KUKA KRL program: MyProgram_165().src

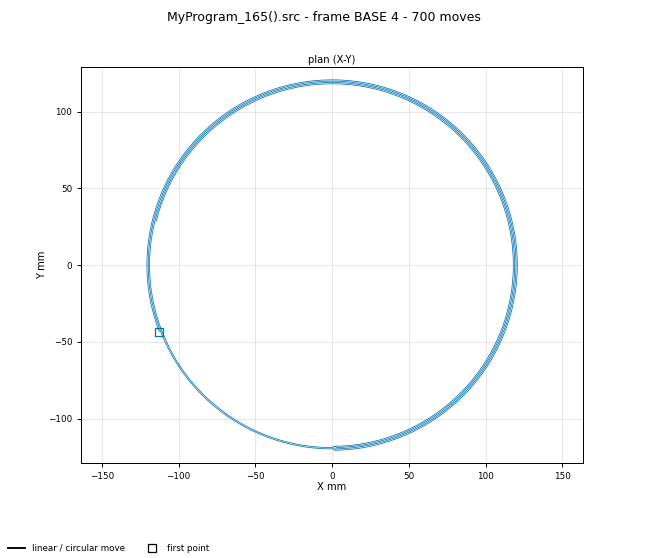
[picture p0: tool path of MyProgram_165().src in frame BASE 4, 700 of 700 moves have a stored position in this frame; points joined in program order, loops and branches not executed]
&ACCESS RVP
&REL 1
&PARAM TEMPLATE = C:\KRC\Roboter\Template\vorgabe
&PARAM EDITMASK = *
DEF MyProgram_165()
; ---- Setting reference (Base) ----
$BASE = BASE_DATA[4]

; --------------------------
; ---- Setting tool (TCP) ----
$TOOL = TOOL_DATA[3]
; --------------------------

$VEL.CP = VEL_APROX_PRINT
Startdeposition()
$VEL.CP = VEL_PRINT
LIN {X -112.6029,Y -43.4357,Z 125,A -162.8947,B 24.9558,C -1.5362,E1 24.8502,E2 249.1159} C_DIS
LIN {X -113.6349,Y -40.6592,Z 125,A -164.31,B 24.9556,C -1.54,E1 24.8489,E2 250.5301} C_DIS
LIN {X -114.5985,Y -37.8582,Z 125,A -165.7254,B 24.9553,C -1.5438,E1 24.8476,E2 251.9444} C_DIS
LIN {X -115.4923,Y -35.0371,Z 125,A -167.1395,B 24.9551,C -1.5477,E1 24.8464,E2 253.3573} C_DIS
LIN {X -116.1833,Y -32.6652,Z 125,A -168.3736,B 24.9551,C -1.5488,E1 24.8455,E2 254.5961} C_DIS
LIN {X -117.0731,Y -29.3253,Z 125,A -169.9721,B 24.9547,C -1.5556,E1 24.8444,E2 256.1875} C_DIS
LIN {X -117.7575,Y -26.4433,Z 125,A -171.3879,B 24.9544,C -1.5596,E1 24.8435,E2 257.6022} C_DIS
LIN {X -118.371,Y -23.5454,Z 125,A -172.8035,B 24.9542,C -1.5637,E1 24.8427,E2 259.0165} C_DIS
LIN {X -118.9131,Y -20.6334,Z 125,A -174.2195,B 24.954,C -1.5677,E1 24.842,E2 260.4313} C_DIS
LIN {X -119.592,Y -16.2425,Z 125,A -176.3434,B 24.9536,C -1.5738,E1 24.8411,E2 262.5532} C_DIS
LIN {X -119.9546,Y -13.3027,Z 125,A -177.7592,B 24.9533,C -1.578,E1 24.8407,E2 263.9677} C_DIS
LIN {X -120.2449,Y -10.3549,Z 125,A -179.1753,B 24.9531,C -1.5821,E1 24.8403,E2 265.3825} C_DIS
LIN {X -120.4629,Y -7.4008,Z 125,A 179.4086,B 24.9529,C -1.5862,E1 24.84,E2 266.7971} C_DIS
LIN {X -120.6082,Y -4.4423,Z 125,A 177.9925,B 24.9526,C -1.5904,E1 24.8399,E2 268.2119} C_DIS
LIN {X -120.6878,Y -0.4383,Z 125,A 176.0198,B 24.9524,C -1.5936,E1 24.8398,E2 270.1888} C_DIS
LIN {X -120.6536,Y 2.9619,Z 125,A 174.4521,B 24.952,C -1.6008,E1 24.8398,E2 271.7488} C_DIS
LIN {X -120.5446,Y 5.922,Z 125,A 173.0359,B 24.9517,C -1.605,E1 24.84,E2 273.1636} C_DIS
LIN {X -120.363,Y 8.8785,Z 125,A 171.6198,B 24.9515,C -1.6091,E1 24.8403,E2 274.5783} C_DIS
LIN {X -120.1088,Y 11.8297,Z 125,A 170.2037,B 24.9512,C -1.6133,E1 24.8407,E2 275.9929} C_DIS
LIN {X -119.7823,Y 14.7737,Z 125,A 168.7876,B 24.951,C -1.6175,E1 24.8411,E2 277.4075} C_DIS
LIN {X -119.2402,Y 18.6372,Z 125,A 166.8598,B 24.9508,C -1.6204,E1 24.8419,E2 279.34} C_DIS
LIN {X -118.651,Y 22.0911,Z 125,A 165.2473,B 24.9503,C -1.6279,E1 24.8427,E2 280.9441} C_DIS
LIN {X -118.0731,Y 24.9963,Z 125,A 163.8312,B 24.9501,C -1.632,E1 24.8435,E2 282.3587} C_DIS
LIN {X -117.4241,Y 27.8864,Z 125,A 162.4152,B 24.9498,C -1.6361,E1 24.8444,E2 283.7732} C_DIS
LIN {X -116.7044,Y 30.7597,Z 125,A 160.9991,B 24.9496,C -1.6402,E1 24.8453,E2 285.1878} C_DIS
LIN {X -115.9143,Y 33.6145,Z 125,A 159.5832,B 24.9493,C -1.6443,E1 24.8464,E2 286.6021} C_DIS
LIN {X -115.1524,Y 36.1334,Z 125,A 158.2993,B 24.9492,C -1.6468,E1 24.8475,E2 287.8873} C_DIS
LIN {X -114.1253,Y 39.2617,Z 125,A 156.7515,B 24.9488,C -1.6524,E1 24.8488,E2 289.4308} C_DIS
LIN {X -113.1274,Y 42.0506,Z 125,A 155.3357,B 24.9486,C -1.6564,E1 24.8502,E2 290.8451} C_DIS
LIN {X -112.0614,Y 44.8143,Z 125,A 153.9202,B 24.9483,C -1.6604,E1 24.8516,E2 292.259} C_DIS
LIN {X -110.9278,Y 47.5509,Z 125,A 152.5045,B 24.9481,C -1.6643,E1 24.8532,E2 293.6731} C_DIS
LIN {X -109.7275,Y 50.2589,Z 125,A 151.089,B 24.9478,C -1.6682,E1 24.8548,E2 295.0871} C_DIS
LIN {X -108.461,Y 52.9366,Z 125,A 149.6737,B 24.9476,C -1.6721,E1 24.8565,E2 296.5009} C_DIS
LIN {X -107.1292,Y 55.5824,Z 125,A 148.2584,B 24.9474,C -1.6759,E1 24.8583,E2 297.9146} C_DIS
LIN {X -105.7329,Y 58.1948,Z 125,A 146.8429,B 24.9471,C -1.6797,E1 24.8602,E2 299.3286} C_DIS
LIN {X -104.2729,Y 60.772,Z 125,A 145.4281,B 24.9469,C -1.6835,E1 24.8621,E2 300.7418} C_DIS
LIN {X -102.75,Y 63.3127,Z 125,A 144.013,B 24.9467,C -1.6871,E1 24.8642,E2 302.1554} C_DIS
LIN {X -101.1653,Y 65.8153,Z 125,A 142.598,B 24.9464,C -1.6908,E1 24.8663,E2 303.5688} C_DIS
LIN {X -99.5197,Y 68.2782,Z 125,A 141.1833,B 24.9462,C -1.6944,E1 24.8685,E2 304.9821} C_DIS
LIN {X -97.8985,Y 70.5815,Z 125,A 139.8326,B 24.946,C -1.6975,E1 24.8707,E2 306.3319} C_DIS
LIN {X -96.0495,Y 73.0791,Z 125,A 138.3539,B 24.9458,C -1.7014,E1 24.8732,E2 307.8084} C_DIS
LIN {X -93.2946,Y 76.5649,Z 125,A 136.233,B 24.9454,C -1.7065,E1 24.8769,E2 309.9271} C_DIS
LIN {X -91.3875,Y 78.8314,Z 125,A 134.8186,B 24.9452,C -1.7099,E1 24.8794,E2 311.34} C_DIS
LIN {X -89.4254,Y 81.0504,Z 125,A 133.4045,B 24.945,C -1.7131,E1 24.8821,E2 312.7527} C_DIS
LIN {X -87.4094,Y 83.2206,Z 125,A 131.9907,B 24.9448,C -1.7163,E1 24.8848,E2 314.1649} C_DIS
LIN {X -85.3407,Y 85.3407,Z 125,A 130.577,B 24.9446,C -1.7195,E1 24.8875,E2 315.5772} C_DIS
LIN {X -83.2206,Y 87.4094,Z 125,A 129.1635,B 24.9444,C -1.7225,E1 24.8904,E2 316.9892} C_DIS
LIN {X -81.0504,Y 89.4254,Z 125,A 127.7501,B 24.9442,C -1.7255,E1 24.8933,E2 318.4012} C_DIS
LIN {X -78.8314,Y 91.3875,Z 125,A 126.3371,B 24.944,C -1.7285,E1 24.8963,E2 319.8128} C_DIS
LIN {X -76.5649,Y 93.2946,Z 125,A 124.9241,B 24.9438,C -1.7313,E1 24.8993,E2 321.2244} C_DIS
LIN {X -74.2523,Y 95.1455,Z 125,A 123.511,B 24.9436,C -1.7341,E1 24.9024,E2 322.6362} C_DIS
LIN {X -71.8949,Y 96.9391,Z 125,A 122.0984,B 24.9435,C -1.7368,E1 24.9055,E2 324.0474} C_DIS
LIN {X -69.4943,Y 98.6743,Z 125,A 120.6859,B 24.9433,C -1.7394,E1 24.9087,E2 325.4586} C_DIS
LIN {X -67.0518,Y 100.3501,Z 125,A 119.2737,B 24.9431,C -1.742,E1 24.912,E2 326.8695} C_DIS
LIN {X -63.7759,Y 102.4607,Z 125,A 117.3526,B 24.9431,C -1.7425,E1 24.9165,E2 328.7955} C_DIS
LIN {X -60.772,Y 104.2729,Z 125,A 115.744,B 24.9427,C -1.7479,E1 24.9204,E2 330.396} C_DIS
LIN {X -57.2872,Y 106.2252,Z 125,A 113.8456,B 24.9425,C -1.7512,E1 24.925,E2 332.292} C_DIS
LIN {X -54.2636,Y 107.8032,Z 125,A 112.2154,B 24.9424,C -1.7534,E1 24.9291,E2 333.9215} C_DIS
LIN {X -51.6016,Y 109.1025,Z 125,A 110.804,B 24.9422,C -1.7554,E1 24.9326,E2 335.3317} C_DIS
LIN {X -48.1374,Y 110.6722,Z 125,A 108.9928,B 24.9421,C -1.7579,E1 24.9372,E2 337.1413} C_DIS
LIN {X -45.4069,Y 111.8202,Z 125,A 107.5823,B 24.942,C -1.7597,E1 24.9409,E2 338.5507} C_DIS
LIN {X -42.3982,Y 112.9958,Z 125,A 106.0121,B 24.942,C -1.7602,E1 24.945,E2 340.1232} C_DIS
LIN {X -39.2617,Y 114.1253,Z 125,A 104.4574,B 24.9417,C -1.7634,E1 24.949,E2 341.6733} C_DIS
LIN {X -36.4491,Y 115.0545,Z 125,A 103.0473,B 24.9417,C -1.7649,E1 24.9528,E2 343.0823} C_DIS
LIN {X -33.6145,Y 115.9143,Z 125,A 101.6376,B 24.9415,C -1.7663,E1 24.9566,E2 344.491} C_DIS
LIN {X -30.7597,Y 116.7044,Z 125,A 100.2283,B 24.9415,C -1.7676,E1 24.9604,E2 345.8993} C_DIS
LIN {X -27.8864,Y 117.4241,Z 125,A 98.8194,B 24.9414,C -1.7689,E1 24.9642,E2 347.3072} C_DIS
LIN {X -24.9963,Y 118.0731,Z 125,A 97.4103,B 24.9413,C -1.77,E1 24.968,E2 348.7155} C_DIS
LIN {X -22.0911,Y 118.651,Z 125,A 96.0017,B 24.9413,C -1.771,E1 24.9719,E2 350.1232} C_DIS
LIN {X -18.3412,Y 119.2859,Z 125,A 94.2227,B 24.941,C -1.7736,E1 24.9768,E2 351.8978} C_DIS
LIN {X -15.4082,Y 119.7001,Z 125,A 92.7653,B 24.9411,C -1.7722,E1 24.9808,E2 353.3596} C_DIS
LIN {X -11.8297,Y 120.1088,Z 125,A 91.073,B 24.9411,C -1.7738,E1 24.9855,E2 355.0489} C_DIS
LIN {X -8.8785,Y 120.363,Z 125,A 89.6655,B 24.941,C -1.7744,E1 24.9894,E2 356.4557} C_DIS
LIN {X -5.922,Y 120.5446,Z 125,A 88.2578,B 24.941,C -1.7749,E1 24.9933,E2 357.8628} C_DIS
LIN {X -1.4811,Y 120.6809,Z 125,A 86.1474,B 24.941,C -1.7754,E1 24.9992,E2 359.9721} C_DIS
LIN {X 1.4811,Y 120.6809,Z 125,A 84.7407,B 24.941,C -1.7757,E1 25.0032,E2 361.3781} C_DIS
LIN {X 4.4423,Y 120.6082,Z 125,A 83.3343,B 24.9409,C -1.7757,E1 25.0071,E2 362.784} C_DIS
LIN {X 7.4008,Y 120.4629,Z 125,A 81.9278,B 24.9409,C -1.7757,E1 25.011,E2 364.1899} C_DIS
LIN {X 10.3549,Y 120.2449,Z 125,A 80.5218,B 24.9409,C -1.7757,E1 25.0149,E2 365.5953} C_DIS
LIN {X 13.3027,Y 119.9546,Z 125,A 79.116,B 24.9409,C -1.7755,E1 25.0188,E2 367.0006} C_DIS
LIN {X 16.2425,Y 119.592,Z 125,A 77.7102,B 24.9409,C -1.7752,E1 25.0227,E2 368.4061} C_DIS
LIN {X 19.1726,Y 119.1574,Z 125,A 76.3051,B 24.9409,C -1.7748,E1 25.0266,E2 369.8107} C_DIS
LIN {X 22.0911,Y 118.651,Z 125,A 74.8999,B 24.9409,C -1.7744,E1 25.0304,E2 371.2155} C_DIS
LIN {X 24.9963,Y 118.0731,Z 125,A 73.4952,B 24.941,C -1.7738,E1 25.0343,E2 372.6198} C_DIS
LIN {X 27.8864,Y 117.4241,Z 125,A 72.0905,B 24.941,C -1.7731,E1 25.0381,E2 374.0243} C_DIS
LIN {X 30.7597,Y 116.7044,Z 125,A 70.6861,B 24.9411,C -1.7723,E1 25.0419,E2 375.4284} C_DIS
LIN {X 33.6145,Y 115.9143,Z 125,A 69.2821,B 24.9411,C -1.7714,E1 25.0457,E2 376.8321} C_DIS
LIN {X 36.4491,Y 115.0545,Z 125,A 67.878,B 24.9413,C -1.7704,E1 25.0494,E2 378.236} C_DIS
LIN {X 38.7619,Y 114.2938,Z 125,A 66.6649,B 24.9415,C -1.7668,E1 25.0527,E2 379.4554} C_DIS
LIN {X 42.0506,Y 113.1274,Z 125,A 65.0709,B 24.9415,C -1.7682,E1 25.0568,E2 381.0428} C_DIS
LIN {X 44.8143,Y 112.0614,Z 125,A 63.6677,B 24.9415,C -1.7669,E1 25.0605,E2 382.446} C_DIS
LIN {X 47.5509,Y 110.9278,Z 125,A 62.2648,B 24.9415,C -1.7655,E1 25.0641,E2 383.8488} C_DIS
LIN {X 50.2589,Y 109.7275,Z 125,A 60.8619,B 24.9417,C -1.764,E1 25.0676,E2 385.2517} C_DIS
LIN {X 52.9366,Y 108.461,Z 125,A 59.4596,B 24.9417,C -1.7625,E1 25.0712,E2 386.654} C_DIS
LIN {X 56.562,Y 106.6133,Z 125,A 57.5008,B 24.942,C -1.7587,E1 25.076,E2 388.6164} C_DIS
LIN {X 59.4879,Y 105.0108,Z 125,A 55.954,B 24.942,C -1.7581,E1 25.0798,E2 390.1599} C_DIS
LIN {X 62.0471,Y 103.5193,Z 125,A 54.5523,B 24.9422,C -1.7563,E1 25.0832,E2 391.5618} C_DIS
LIN {X 64.3587,Y 102.0967,Z 125,A 53.2527,B 24.9424,C -1.7538,E1 25.0863,E2 392.8631} C_DIS
LIN {X 67.0518,Y 100.3501,Z 125,A 51.7493,B 24.9424,C -1.7522,E1 25.0898,E2 394.3652} C_DIS
LIN {X 69.4943,Y 98.6743,Z 125,A 50.3482,B 24.9426,C -1.7501,E1 25.093,E2 395.7666} C_DIS
LIN {X 71.6715,Y 97.1027,Z 125,A 49.0595,B 24.9428,C -1.7472,E1 25.0959,E2 397.0575} C_DIS
LIN {X 74.2523,Y 95.1455,Z 125,A 47.5463,B 24.9428,C -1.7455,E1 25.0992,E2 398.5691} C_DIS
LIN {X 76.5649,Y 93.2946,Z 125,A 46.1458,B 24.9431,C -1.7431,E1 25.1023,E2 399.97} C_DIS
LIN {X 78.5212,Y 91.6518,Z 125,A 44.9007,B 24.9433,C -1.7392,E1 25.1049,E2 401.2194} C_DIS
LIN {X 81.0504,Y 89.4254,Z 125,A 43.3453,B 24.9433,C -1.7381,E1 25.1082,E2 402.7713} C_DIS
LIN {X 83.2206,Y 87.4094,Z 125,A 41.9454,B 24.9436,C -1.7354,E1 25.111,E2 404.1718} C_DIS
LIN {X 85.3407,Y 85.3407,Z 125,A 40.5457,B 24.9437,C -1.7327,E1 25.1138,E2 405.572} C_DIS
LIN {X 87.4094,Y 83.2206,Z 125,A 39.146,B 24.9439,C -1.7299,E1 25.1165,E2 406.9723} C_DIS
LIN {X 89.4086,Y 81.0687,Z 125,A 37.758,B 24.9441,C -1.7271,E1 25.1191,E2 408.3609} C_DIS
LIN {X 91.3875,Y 78.8314,Z 125,A 36.3474,B 24.9443,C -1.7241,E1 25.1217,E2 409.7721} C_DIS
LIN {X 93.2946,Y 76.5649,Z 125,A 34.948,B 24.9445,C -1.7211,E1 25.1242,E2 411.1721} C_DIS
LIN {X 95.1455,Y 74.2523,Z 125,A 33.5493,B 24.9447,C -1.718,E1 25.1267,E2 412.5716} C_DIS
LIN {X 96.9391,Y 71.8949,Z 125,A 32.1503,B 24.9449,C -1.7149,E1 25.129,E2 413.9713} C_DIS
LIN {X 98.6743,Y 69.4943,Z 125,A 30.7518,B 24.9451,C -1.7117,E1 25.1313,E2 415.3705} C_DIS
LIN {X 100.3501,Y 67.0518,Z 125,A 29.3533,B 24.9453,C -1.7084,E1 25.1335,E2 416.7699} C_DIS
LIN {X 101.9654,Y 64.5689,Z 125,A 27.9547,B 24.9455,C -1.7051,E1 25.1356,E2 418.1693} C_DIS
LIN {X 103.3302,Y 62.3582,Z 125,A 26.6977,B 24.9458,C -1.7007,E1 25.1374,E2 419.4303} C_DIS
LIN {X 105.0108,Y 59.4879,Z 125,A 25.1587,B 24.946,C -1.6983,E1 25.1396,E2 420.967} C_DIS
LIN {X 106.4391,Y 56.8929,Z 125,A 23.7606,B 24.9462,C -1.6948,E1 25.1414,E2 422.3661} C_DIS
LIN {X 107.8032,Y 54.2636,Z 125,A 22.3629,B 24.9464,C -1.6912,E1 25.1432,E2 423.7647} C_DIS
LIN {X 109.1025,Y 51.6016,Z 125,A 20.9651,B 24.9466,C -1.6876,E1 25.1449,E2 425.1635} C_DIS
LIN {X 110.336,Y 48.9086,Z 125,A 19.5676,B 24.9469,C -1.684,E1 25.1465,E2 426.562} C_DIS
LIN {X 111.503,Y 46.1861,Z 125,A 18.1699,B 24.9471,C -1.6803,E1 25.148,E2 427.9608} C_DIS
LIN {X 112.5558,Y 43.5555,Z 125,A 16.829,B 24.9473,C -1.6765,E1 25.1494,E2 429.3032} C_DIS
LIN {X 113.588,Y 40.788,Z 125,A 15.4352,B 24.9476,C -1.6727,E1 25.1507,E2 430.6981} C_DIS
LIN {X 114.5985,Y 37.8582,Z 125,A 13.978,B 24.9478,C -1.6689,E1 25.152,E2 432.1559} C_DIS
LIN {X 115.4931,Y 35.0344,Z 125,A 12.5811,B 24.948,C -1.6651,E1 25.1532,E2 433.554} C_DIS
LIN {X 116.3181,Y 32.1896,Z 125,A 11.184,B 24.9483,C -1.6612,E1 25.1543,E2 434.9522} C_DIS
LIN {X 117.0731,Y 29.3253,Z 125,A 9.787,B 24.9485,C -1.6573,E1 25.1552,E2 436.3504} C_DIS
LIN {X 117.7575,Y 26.4433,Z 125,A 8.3902,B 24.9488,C -1.6533,E1 25.1561,E2 437.7485} C_DIS
LIN {X 118.371,Y 23.5454,Z 125,A 6.9934,B 24.949,C -1.6493,E1 25.1569,E2 439.1465} C_DIS
LIN {X 118.9131,Y 20.6334,Z 125,A 5.5965,B 24.9493,C -1.6453,E1 25.1576,E2 440.5447} C_DIS
LIN {X 119.3837,Y 17.7089,Z 125,A 4.2001,B 24.9495,C -1.6413,E1 25.1582,E2 441.9423} C_DIS
LIN {X 119.7823,Y 14.7737,Z 125,A 2.8031,B 24.9498,C -1.6372,E1 25.1587,E2 443.3406} C_DIS
LIN {X 120.1088,Y 11.8297,Z 125,A 1.4066,B 24.95,C -1.6332,E1 25.1591,E2 444.7385} C_DIS
LIN {X 120.363,Y 8.8785,Z 125,A 0.0101,B 24.9503,C -1.6291,E1 25.1594,E2 446.1363} C_DIS
LIN {X 120.5446,Y 5.922,Z 125,A -1.3868,B 24.9505,C -1.625,E1 25.1596,E2 447.5346} C_DIS
LIN {X 120.6809,Y 1.481,Z 125,A -3.6105,B 24.9513,C -1.6125,E1 25.1598,E2 449.7746} C_DIS
LIN {X 120.6536,Y -2.9619,Z 125,A -5.5761,B 24.9513,C -1.6127,E1 25.1598,E2 451.728} C_DIS
LIN {X 120.5446,Y -5.922,Z 125,A -6.9725,B 24.9515,C -1.6085,E1 25.1595,E2 453.1259} C_DIS
LIN {X 120.363,Y -8.8785,Z 125,A -8.369,B 24.9518,C -1.6044,E1 25.1593,E2 454.5238} C_DIS
LIN {X 120.1088,Y -11.8297,Z 125,A -9.7654,B 24.952,C -1.6003,E1 25.1589,E2 455.9217} C_DIS
LIN {X 119.7823,Y -14.7737,Z 125,A -11.1618,B 24.9523,C -1.5962,E1 25.1585,E2 457.3195} C_DIS
LIN {X 119.3837,Y -17.7089,Z 125,A -12.5582,B 24.9525,C -1.592,E1 25.1579,E2 458.7173} C_DIS
LIN {X 118.9131,Y -20.6334,Z 125,A -13.955,B 24.9528,C -1.5879,E1 25.1573,E2 460.1156} C_DIS
LIN {X 118.371,Y -23.5454,Z 125,A -15.3514,B 24.953,C -1.5838,E1 25.1565,E2 461.5136} C_DIS
LIN {X 117.5681,Y -27.263,Z 125,A -17.1815,B 24.9534,C -1.5768,E1 25.1554,E2 463.3496} C_DIS
LIN {X 116.7044,Y -30.7597,Z 125,A -18.843,B 24.9536,C -1.5737,E1 25.1543,E2 465.0089} C_DIS
LIN {X 115.9143,Y -33.6145,Z 125,A -20.2397,B 24.9538,C -1.5696,E1 25.1532,E2 466.4072} C_DIS
LIN {X 115.0545,Y -36.4491,Z 125,A -21.6363,B 24.9541,C -1.5656,E1 25.1521,E2 467.8053} C_DIS
LIN {X 114.1253,Y -39.2617,Z 125,A -23.0331,B 24.9543,C -1.5616,E1 25.1508,E2 469.2036} C_DIS
LIN {X 113.1274,Y -42.0506,Z 125,A -24.43,B 24.9545,C -1.5576,E1 25.1495,E2 470.602} C_DIS
LIN {X 112.0614,Y -44.8143,Z 125,A -25.8269,B 24.9548,C -1.5537,E1 25.1481,E2 472.0005} C_DIS
LIN {X 111.1126,Y -47.1124,Z 125,A -27.0487,B 24.9551,C -1.548,E1 25.1467,E2 473.2289} C_DIS
LIN {X 109.7275,Y -50.2589,Z 125,A -28.621,B 24.9552,C -1.5459,E1 25.1449,E2 474.7976} C_DIS
LIN {X 108.5122,Y -52.8301,Z 125,A -29.9662,B 24.9554,C -1.5421,E1 25.1433,E2 476.1447} C_DIS
LIN {X 107.1309,Y -55.5791,Z 125,A -31.4135,B 24.9557,C -1.5383,E1 25.1415,E2 477.5932} C_DIS
LIN {X 105.7329,Y -58.1948,Z 125,A -32.8128,B 24.9559,C -1.5345,E1 25.1396,E2 478.994} C_DIS
LIN {X 104.4838,Y -60.405,Z 125,A -34.0505,B 24.9562,C -1.5294,E1 25.1379,E2 480.2374} C_DIS
LIN {X 102.75,Y -63.3127,Z 125,A -35.6077,B 24.9563,C -1.5271,E1 25.1356,E2 481.792} C_DIS
LIN {X 101.1653,Y -65.8153,Z 125,A -37.0055,B 24.9565,C -1.5235,E1 25.1335,E2 483.1913} C_DIS
LIN {X 99.5795,Y -68.1898,Z 125,A -38.3561,B 24.9567,C -1.5199,E1 25.1314,E2 484.5437} C_DIS
LIN {X 97.8141,Y -70.6999,Z 125,A -39.8011,B 24.9569,C -1.5164,E1 25.1291,E2 485.9899} C_DIS
LIN {X 96.0495,Y -73.0791,Z 125,A -41.1992,B 24.9571,C -1.513,E1 25.1267,E2 487.3895} C_DIS
LIN {X 94.2272,Y -75.4143,Z 125,A -42.5975,B 24.9573,C -1.5095,E1 25.1243,E2 488.7893} C_DIS
LIN {X 92.348,Y -77.704,Z 125,A -43.9957,B 24.9575,C -1.5062,E1 25.1218,E2 490.1891} C_DIS
LIN {X 90.4133,Y -79.947,Z 125,A -45.394,B 24.9577,C -1.5029,E1 25.1192,E2 491.5888} C_DIS
LIN {X 88.5029,Y -82.0557,Z 125,A -46.741,B 24.9579,C -1.4996,E1 25.1167,E2 492.9375} C_DIS
LIN {X 85.6291,Y -85.0488,Z 125,A -48.7349,B 24.9582,C -1.4935,E1 25.1128,E2 494.9372} C_DIS
LIN {X 83.2206,Y -87.4094,Z 125,A -50.2897,B 24.9583,C -1.4919,E1 25.1097,E2 496.4896} C_DIS
LIN {X 81.0504,Y -89.4254,Z 125,A -51.6888,B 24.9585,C -1.4889,E1 25.1068,E2 497.8901} C_DIS
LIN {X 78.8314,Y -91.3875,Z 125,A -53.0878,B 24.9586,C -1.4859,E1 25.1039,E2 499.2904} C_DIS
LIN {X 76.5649,Y -93.2946,Z 125,A -54.4874,B 24.9588,C -1.4831,E1 25.1009,E2 500.6915} C_DIS
LIN {X 74.2523,Y -95.1455,Z 125,A -55.8872,B 24.9589,C -1.4803,E1 25.0978,E2 502.0926} C_DIS
LIN {X 71.8949,Y -96.9391,Z 125,A -57.2871,B 24.9591,C -1.4776,E1 25.0947,E2 503.4938} C_DIS
LIN {X 68.8035,Y -99.1545,Z 125,A -59.0847,B 24.9593,C -1.4742,E1 25.0906,E2 505.2931} C_DIS
LIN {X 66.22,Y -100.8985,Z 125,A -60.6092,B 24.9596,C -1.4691,E1 25.087,E2 506.8247} C_DIS
LIN {X 63.3127,Y -102.75,Z 125,A -62.188,B 24.9596,C -1.4687,E1 25.0833,E2 508.3994} C_DIS
LIN {X 60.772,Y -104.2729,Z 125,A -63.5886,B 24.9597,C -1.4663,E1 25.0799,E2 509.8013} C_DIS
LIN {X 58.1948,Y -105.7329,Z 125,A -64.9894,B 24.9598,C -1.4641,E1 25.0765,E2 511.2032} C_DIS
LIN {X 55.6548,Y -107.0911,Z 125,A -66.3537,B 24.96,C -1.4618,E1 25.0731,E2 512.5689} C_DIS
LIN {X 52.9366,Y -108.461,Z 125,A -67.7918,B 24.96,C -1.4598,E1 25.0695,E2 514.0081} C_DIS
LIN {X 50.2589,Y -109.7275,Z 125,A -69.1933,B 24.9602,C -1.4578,E1 25.066,E2 515.4108} C_DIS
LIN {X 47.5509,Y -110.9278,Z 125,A -70.5949,B 24.9602,C -1.4558,E1 25.0624,E2 516.8136} C_DIS
LIN {X 44.8143,Y -112.0614,Z 125,A -71.997,B 24.9604,C -1.454,E1 25.0587,E2 518.2167} C_DIS
LIN {X 42.0506,Y -113.1274,Z 125,A -73.399,B 24.9604,C -1.4523,E1 25.0551,E2 519.6199} C_DIS
LIN {X 39.2617,Y -114.1253,Z 125,A -74.8012,B 24.9606,C -1.4506,E1 25.0514,E2 521.0231} C_DIS
LIN {X 36.5066,Y -115.0359,Z 125,A -76.1764,B 24.9606,C -1.449,E1 25.0477,E2 522.3995} C_DIS
LIN {X 33.6145,Y -115.9143,Z 125,A -77.6068,B 24.9607,C -1.4476,E1 25.0439,E2 523.8308} C_DIS
LIN {X 30.7597,Y -116.7044,Z 125,A -79.0098,B 24.9608,C -1.4462,E1 25.0401,E2 525.2348} C_DIS
LIN {X 27.8864,Y -117.4241,Z 125,A -80.4128,B 24.9608,C -1.445,E1 25.0363,E2 526.6387} C_DIS
LIN {X 25.2346,Y -118.0211,Z 125,A -81.713,B 24.961,C -1.4433,E1 25.0328,E2 527.9411} C_DIS
LIN {X 22.0911,Y -118.651,Z 125,A -83.2201,B 24.961,C -1.4427,E1 25.0286,E2 529.4478} C_DIS
LIN {X 19.1726,Y -119.1574,Z 125,A -84.6243,B 24.961,C -1.4417,E1 25.0248,E2 530.8529} C_DIS
LIN {X 16.2425,Y -119.592,Z 125,A -86.0283,B 24.9611,C -1.4409,E1 25.0209,E2 532.2577} C_DIS
LIN {X 13.3027,Y -119.9546,Z 125,A -87.4326,B 24.9611,C -1.4401,E1 25.017,E2 533.6629} C_DIS
LIN {X 10.3549,Y -120.2449,Z 125,A -88.8372,B 24.9611,C -1.4394,E1 25.0131,E2 535.0682} C_DIS
LIN {X 7.4008,Y -120.4629,Z 125,A -90.2421,B 24.9612,C -1.4388,E1 25.0092,E2 536.4739} C_DIS
LIN {X 4.6043,Y -120.6012,Z 125,A -91.5771,B 24.9612,C -1.4381,E1 25.0054,E2 537.8103} C_DIS
LIN {X 1.4811,Y -120.6809,Z 125,A -93.0526,B 24.9612,C -1.438,E1 25.0013,E2 539.2857} C_DIS
LIN {X 1.4811,Y -120.6809,Z 125,A -93.0526,B 24.9612,C -1.438,E1 25.0013,E2 539.2857} C_DIS
Enddeposition()
LIN {X 0.8495,Y -119.8203,Z 125,A -93.2213,B 24.9601,C -1.4593,E1 25.001,E2 539.4041} C_DIS
Startdeposition()
$VEL.CP = VEL_PRINT
LIN {X 5.6082,Y -119.6935,Z 125,A -90.3947,B 24.9587,C -1.4855,E1 25.0091,E2 536.5158} C_DIS
LIN {X 9.4036,Y -119.4544,Z 125,A -88.6242,B 24.9587,C -1.4841,E1 25.014,E2 534.7494} C_DIS
LIN {X 12.515,Y -119.1685,Z 125,A -87.1094,B 24.9587,C -1.4859,E1 25.0182,E2 533.2313} C_DIS
LIN {X 16.0428,Y -118.7469,Z 125,A -85.3137,B 24.9583,C -1.4916,E1 25.0232,E2 531.4237} C_DIS
LIN {X 19.8544,Y -118.1676,Z 125,A -83.6129,B 24.9586,C -1.4862,E1 25.0278,E2 529.7372} C_DIS
LIN {X 23.2177,Y -117.5544,Z 125,A -81.8254,B 24.9581,C -1.4948,E1 25.0328,E2 527.9314} C_DIS
LIN {X 27.1102,Y -116.7168,Z 125,A -80.0364,B 24.9583,C -1.4912,E1 25.0376,E2 526.1534} C_DIS
LIN {X 30.7989,Y -115.799,Z 125,A -78.211,B 24.9583,C -1.4934,E1 25.0426,E2 524.3256} C_DIS
LIN {X 34.222,Y -114.8331,Z 125,A -76.6065,B 24.9583,C -1.4908,E1 25.0468,E2 522.7301} C_DIS
LIN {X 36.9667,Y -113.9791,Z 125,A -75.2801,B 24.9583,C -1.4902,E1 25.0504,E2 521.4076} C_DIS
LIN {X 39.7283,Y -113.0461,Z 125,A -73.8848,B 24.9583,C -1.492,E1 25.0541,E2 520.0106} C_DIS
LIN {X 42.0511,Y -112.2035,Z 125,A -72.401,B 24.9574,C -1.5081,E1 25.058,E2 518.492} C_DIS
LIN {X 45.74,Y -110.7519,Z 125,A -70.609,B 24.9575,C -1.5058,E1 25.0626,E2 516.7094} C_DIS
LIN {X 49.2968,Y -109.2135,Z 125,A -68.852,B 24.9576,C -1.5041,E1 25.0671,E2 514.9609} C_DIS
LIN {X 52.6411,Y -107.6434,Z 125,A -67.103,B 24.9576,C -1.5061,E1 25.0715,E2 513.2117} C_DIS
LIN {X 55.6557,Y -106.1143,Z 125,A -64.8703,B 24.9556,C -1.5388,E1 25.0772,E2 510.9079} C_DIS
LIN {X 59.6674,Y -103.9113,Z 125,A -63.3368,B 24.9572,C -1.5109,E1 25.0808,E2 509.4449} C_DIS
LIN {X 63.2461,Y -101.7731,Z 125,A -61.2756,B 24.9568,C -1.518,E1 25.0857,E2 507.3734} C_DIS
LIN {X 66.1821,Y -99.8888,Z 125,A -59.5906,B 24.9566,C -1.5221,E1 25.0897,E2 505.6843} C_DIS
LIN {X 68.4808,Y -98.3268,Z 125,A -58.1034,B 24.956,C -1.5325,E1 25.0931,E2 504.1775} C_DIS
LIN {X 72.9915,Y -95.0265,Z 125,A -55.6577,B 24.9563,C -1.5272,E1 25.0985,E2 501.7533} C_DIS
LIN {X 76.1963,Y -92.4778,Z 125,A -53.8788,B 24.9566,C -1.5228,E1 25.1024,E2 499.9914} C_DIS
LIN {X 80.4851,Y -88.7718,Z 125,A -50.2283,B 24.9535,C -1.5753,E1 25.1102,E2 496.2313} C_DIS
LIN {X 84.3813,Y -85.0742,Z 125,A -48.5685,B 24.9558,C -1.5368,E1 25.1133,E2 494.6694} C_DIS
LIN {X 88.1633,Y -81.1482,Z 125,A -45.4332,B 24.9538,C -1.5694,E1 25.1195,E2 491.4708} C_DIS
LIN {X 90.7689,Y -78.2255,Z 125,A -43.9347,B 24.9546,C -1.5558,E1 25.1221,E2 490.0112} C_DIS
LIN {X 93.5303,Y -74.9021,Z 125,A -41.8796,B 24.9544,C -1.5608,E1 25.1258,E2 487.9538} C_DIS
LIN {X 95.7578,Y -72.0292,Z 125,A -40.1765,B 24.9542,C -1.5639,E1 25.1286,E2 486.2516} C_DIS
LIN {X 98.3058,Y -68.511,Z 125,A -38.1047,B 24.9539,C -1.5694,E1 25.132,E2 484.1768} C_DIS
LIN {X 100.5686,Y -65.1458,Z 125,A -35.5438,B 24.9517,C -1.6059,E1 25.136,E2 481.5427} C_DIS
LIN {X 103.1659,Y -60.9472,Z 125,A -34.069,B 24.9539,C -1.5687,E1 25.138,E2 480.1631} C_DIS
LIN {X 104.8675,Y -57.9727,Z 125,A -32.315,B 24.9533,C -1.5793,E1 25.1404,E2 478.3934} C_DIS
LIN {X 106.6324,Y -54.6564,Z 125,A -30.4687,B 24.9528,C -1.5871,E1 25.1428,E2 476.5382} C_DIS
LIN {X 108.3626,Y -51.1441,Z 125,A -28.5753,B 24.9524,C -1.5939,E1 25.1451,E2 474.6391} C_DIS
LIN {X 109.5838,Y -48.4722,Z 125,A -26.9898,B 24.9516,C -1.6072,E1 25.147,E2 473.031} C_DIS
LIN {X 111.4311,Y -44.0561,Z 125,A -24.8386,B 24.9516,C -1.6075,E1 25.1492,E2 470.8909} C_DIS
LIN {X 112.8821,Y -40.1957,Z 125,A -22.985,B 24.9516,C -1.6078,E1 25.151,E2 469.0469} C_DIS
LIN {X 113.9914,Y -36.9288,Z 125,A -21.353,B 24.9513,C -1.6121,E1 25.1524,E2 467.4139} C_DIS
LIN {X 114.9879,Y -33.7001,Z 125,A -19.7906,B 24.9511,C -1.6146,E1 25.1537,E2 465.8545} C_DIS
LIN {X 115.982,Y -30.1003,Z 125,A -17.8641,B 24.9504,C -1.6274,E1 25.1551,E2 463.909} C_DIS
LIN {X 116.986,Y -25.9268,Z 125,A -15.9103,B 24.9503,C -1.6291,E1 25.1563,E2 461.9625} C_DIS
LIN {X 117.6031,Y -22.9644,Z 125,A -14.4732,B 24.95,C -1.6333,E1 25.1571,E2 460.5238} C_DIS
LIN {X 118.1676,Y -19.8542,Z 125,A -12.9283,B 24.9496,C -1.6399,E1 25.1578,E2 458.9725} C_DIS
LIN {X 118.7989,Y -15.6414,Z 125,A -10.9782,B 24.9495,C -1.6422,E1 25.1586,E2 457.0284} C_DIS
LIN {X 119.21,Y -12.1186,Z 125,A -9.4058,B 24.9495,C -1.6417,E1 25.1591,E2 455.4666} C_DIS
LIN {X 119.5911,Y -7.4889,Z 125,A -7.1397,B 24.9489,C -1.6511,E1 25.1595,E2 453.1916} C_DIS
LIN {X 119.8036,Y -2.2047,Z 125,A -4.6025,B 24.9484,C -1.6598,E1 25.1598,E2 450.649} C_DIS
LIN {X 119.7999,Y 2.4043,Z 125,A -2.2761,B 24.9475,C -1.6731,E1 25.1598,E2 448.3052} C_DIS
LIN {X 119.656,Y 6.3457,Z 125,A -0.4589,B 24.9474,C -1.6758,E1 25.1595,E2 446.4924} C_DIS
LIN {X 119.3691,Y 10.4458,Z 125,A 1.5002,B 24.947,C -1.6819,E1 25.1591,E2 444.5306} C_DIS
LIN {X 119.035,Y 13.729,Z 125,A 3.0088,B 24.9469,C -1.6835,E1 25.1586,E2 443.027} C_DIS
LIN {X 118.6119,Y 16.9999,Z 125,A 4.5707,B 24.9466,C -1.6879,E1 25.158,E2 441.4642} C_DIS
LIN {X 117.9931,Y 20.8689,Z 125,A 6.4231,B 24.9463,C -1.6928,E1 25.1571,E2 439.6111} C_DIS
LIN {X 117.359,Y 24.1792,Z 125,A 8.0499,B 24.9459,C -1.6986,E1 25.1563,E2 437.9799} C_DIS
LIN {X 116.5436,Y 27.851,Z 125,A 9.8747,B 24.9455,C -1.7056,E1 25.1551,E2 436.1495} C_DIS
LIN {X 115.7473,Y 30.9902,Z 125,A 11.3309,B 24.9455,C -1.7058,E1 25.1541,E2 434.701} C_DIS
LIN {X 114.8458,Y 34.1792,Z 125,A 13.5927,B 24.943,C -1.7443,E1 25.1522,E2 432.3613} C_DIS
LIN {X 113.3629,Y 38.8191,Z 125,A 15.3619,B 24.9443,C -1.7235,E1 25.1507,E2 430.6512} C_DIS
LIN {X 111.4097,Y 44.1107,Z 125,A 17.9887,B 24.944,C -1.7281,E1 25.1481,E2 428.0282} C_DIS
LIN {X 109.8805,Y 47.7918,Z 125,A 19.8506,B 24.9438,C -1.7315,E1 25.1461,E2 426.1685} C_DIS
LIN {X 108.3864,Y 51.093,Z 125,A 21.6837,B 24.9432,C -1.7414,E1 25.1439,E2 424.322} C_DIS
LIN {X 106.8022,Y 54.324,Z 125,A 23.2552,B 24.9433,C -1.739,E1 25.1419,E2 422.7646} C_DIS
LIN {X 105.1451,Y 57.4666,Z 125,A 25.47,B 24.9413,C -1.769,E1 25.1389,E2 420.4904} C_DIS
LIN {X 103.0902,Y 61.0753,Z 125,A 26.9697,B 24.9426,C -1.7505,E1 25.1369,E2 419.0421} C_DIS
LIN {X 101.1772,Y 64.1976,Z 125,A 28.7384,B 24.9422,C -1.756,E1 25.1342,E2 417.2693} C_DIS
LIN {X 98.965,Y 67.5566,Z 125,A 30.6753,B 24.9418,C -1.7617,E1 25.1312,E2 415.3287} C_DIS
LIN {X 96.7654,Y 70.6699,Z 125,A 32.3796,B 24.9419,C -1.7606,E1 25.1285,E2 413.6353} C_DIS
LIN {X 94.5299,Y 73.6359,Z 125,A 34.0661,B 24.9419,C -1.7606,E1 25.1256,E2 411.9567} C_DIS
LIN {X 92.4515,Y 76.2279,Z 125,A 35.7757,B 24.9413,C -1.7703,E1 25.1226,E2 410.2322} C_DIS
LIN {X 90.2172,Y 78.8582,Z 125,A 37.3204,B 24.9413,C -1.7691,E1 25.1198,E2 408.6974} C_DIS
LIN {X 88.0336,Y 81.2895,Z 125,A 39.0088,B 24.9407,C -1.7787,E1 25.1166,E2 406.9937} C_DIS
LIN {X 85.3304,Y 84.122,Z 125,A 40.7801,B 24.9407,C -1.7779,E1 25.1131,E2 405.2318} C_DIS
LIN {X 82.7474,Y 86.6657,Z 125,A 42.53,B 24.9405,C -1.7824,E1 25.1096,E2 403.4787} C_DIS
LIN {X 79.9295,Y 89.2694,Z 125,A 44.362,B 24.9402,C -1.7861,E1 25.1058,E2 401.6454} C_DIS
LIN {X 76.9969,Y 91.8125,Z 125,A 46.2839,B 24.9398,C -1.7928,E1 25.1017,E2 399.715} C_DIS
LIN {X 74.1014,Y 94.1638,Z 125,A 48.0336,B 24.9396,C -1.7946,E1 25.0979,E2 397.9677} C_DIS
LIN {X 70.842,Y 96.6394,Z 125,A 49.9002,B 24.9396,C -1.7938,E1 25.0938,E2 396.1097} C_DIS
LIN {X 68.2712,Y 98.4725,Z 125,A 51.5528,B 24.9391,C -1.8032,E1 25.0899,E2 394.4406} C_DIS
LIN {X 65.0133,Y 100.6536,Z 125,A 53.2911,B 24.9393,C -1.7997,E1 25.0859,E2 392.7162} C_DIS
LIN {X 59.8142,Y 103.827,Z 125,A 56.3172,B 24.9386,C -1.8095,E1 25.0786,E2 389.6764} C_DIS
LIN {X 55.9168,Y 105.9768,Z 125,A 58.245,B 24.9391,C -1.8029,E1 25.074,E2 387.7697} C_DIS
LIN {X 53.0091,Y 107.4609,Z 125,A 59.8711,B 24.9387,C -1.808,E1 25.0699,E2 386.136} C_DIS
LIN {X 49.7965,Y 108.9884,Z 125,A 61.6526,B 24.9383,C -1.8138,E1 25.0653,E2 384.3453} C_DIS
LIN {X 46.3589,Y 110.4928,Z 125,A 64.1721,B 24.9358,C -1.8501,E1 25.0587,E2 381.7458} C_DIS
LIN {X 41.2415,Y 112.503,Z 125,A 65.9618,B 24.9384,C -1.813,E1 25.0542,E2 380.0477} C_DIS
LIN {X 38.139,Y 113.5923,Z 125,A 67.7067,B 24.9377,C -1.8224,E1 25.0495,E2 378.2839} C_DIS
LIN {X 34.2541,Y 114.8236,Z 125,A 69.5105,B 24.9381,C -1.8172,E1 25.0448,E2 376.4959} C_DIS
LIN {X 30.4599,Y 115.8895,Z 125,A 71.4783,B 24.9378,C -1.8223,E1 25.0394,E2 374.5191} C_DIS
LIN {X 26.8116,Y 116.7858,Z 125,A 73.1822,B 24.938,C -1.819,E1 25.0348,E2 372.8253} C_DIS
LIN {X 22.8532,Y 117.6246,Z 125,A 74.9875,B 24.9383,C -1.8139,E1 25.0299,E2 371.0343} C_DIS
LIN {X 20.3223,Y 118.0893,Z 125,A 76.4127,B 24.9377,C -1.8233,E1 25.026,E2 369.5884} C_DIS
LIN {X 17.0576,Y 118.6037,Z 125,A 77.9763,B 24.9377,C -1.823,E1 25.0217,E2 368.0269} C_DIS
LIN {X 13.2045,Y 119.0963,Z 125,A 79.8943,B 24.9375,C -1.8261,E1 25.0163,E2 366.1029} C_DIS
LIN {X 9.6338,Y 119.436,Z 125,A 81.4745,B 24.9379,C -1.8201,E1 25.012,E2 364.5379} C_DIS
LIN {X 6.1151,Y 119.6688,Z 125,A 83.2797,B 24.9375,C -1.8256,E1 25.0069,E2 362.7205} C_DIS
LIN {X 2.4958,Y 119.7982,Z 125,A 84.9501,B 24.9377,C -1.8226,E1 25.0023,E2 361.0575} C_DIS
LIN {X -0.7434,Y 119.8216,Z 125,A 86.506,B 24.9377,C -1.8226,E1 24.9979,E2 359.5016} C_DIS
LIN {X -4.8089,Y 119.7278,Z 125,A 88.4227,B 24.9379,C -1.8207,E1 24.9926,E2 357.5891} C_DIS
LIN {X -7.8924,Y 119.5638,Z 125,A 89.8249,B 24.9381,C -1.8168,E1 24.9887,E2 356.1957} C_DIS
LIN {X -11.0467,Y 119.3136,Z 125,A 91.3673,B 24.9381,C -1.8174,E1 24.9844,E2 354.6511} C_DIS
LIN {X -14.6008,Y 118.9329,Z 125,A 93.0717,B 24.9381,C -1.8162,E1 24.9797,E2 352.9485} C_DIS
LIN {X -18.1066,Y 118.4481,Z 125,A 94.8145,B 24.9381,C -1.8174,E1 24.9748,E2 351.2015} C_DIS
LIN {X -22.0022,Y 117.7884,Z 125,A 96.798,B 24.9379,C -1.8201,E1 24.9694,E2 349.2094} C_DIS
LIN {X -25.8236,Y 117.0085,Z 125,A 98.6022,B 24.9382,C -1.8158,E1 24.9645,E2 347.4133} C_DIS
LIN {X -29.4146,Y 116.1582,Z 125,A 100.4659,B 24.938,C -1.8185,E1 24.9594,E2 345.5406} C_DIS
LIN {X -33.6734,Y 114.9958,Z 125,A 102.5142,B 24.9384,C -1.8135,E1 24.9539,E2 343.501} C_DIS
LIN {X -37.3492,Y 113.8553,Z 125,A 104.3268,B 24.9386,C -1.81,E1 24.9491,E2 341.6932} C_DIS
LIN {X -40.503,Y 112.7724,Z 125,A 106.1067,B 24.9382,C -1.8162,E1 24.9444,E2 339.8952} C_DIS
LIN {X -44.8577,Y 111.111,Z 125,A 108.1903,B 24.9388,C -1.8068,E1 24.939,E2 337.8296} C_DIS
LIN {X -47.8523,Y 109.8541,Z 125,A 110.3169,B 24.9372,C -1.8299,E1 24.9334,E2 335.6429} C_DIS
LIN {X -52.0896,Y 107.9096,Z 125,A 111.9501,B 24.9393,C -1.8,E1 24.9295,E2 334.0767} C_DIS
LIN {X -55.7599,Y 106.0594,Z 125,A 113.9085,B 24.9395,C -1.7964,E1 24.9246,E2 332.1215} C_DIS
LIN {X -58.2484,Y 104.7135,Z 125,A 115.4971,B 24.939,C -1.8044,E1 24.9207,E2 330.5094} C_DIS
LIN {X -62.1661,Y 102.436,Z 125,A 117.4231,B 24.94,C -1.7898,E1 24.9161,E2 328.6121} C_DIS
LIN {X -65.07,Y 100.6173,Z 125,A 119.0659,B 24.9402,C -1.7869,E1 24.9122,E2 326.9711} C_DIS
LIN {X -67.5985,Y 98.9366,Z 125,A 121.3705,B 24.9378,C -1.8214,E1 24.9068,E2 324.5766} C_DIS
LIN {X -72.1212,Y 95.6887,Z 125,A 123.4171,B 24.94,C -1.7887,E1 24.9023,E2 322.6004} C_DIS
LIN {X -75.7736,Y 92.824,Z 125,A 125.419,B 24.941,C -1.7744,E1 24.898,E2 320.6252} C_DIS
LIN {X -79.4193,Y 89.7261,Z 125,A 127.7119,B 24.9413,C -1.7694,E1 24.8932,E2 318.3352} C_DIS
LIN {X -81.8543,Y 87.5085,Z 125,A 129.1428,B 24.942,C -1.7595,E1 24.8903,E2 316.9221} C_DIS
LIN {X -84.494,Y 84.9628,Z 125,A 131.1245,B 24.9416,C -1.765,E1 24.8863,E2 314.9188} C_DIS
LIN {X -86.4136,Y 83.009,Z 125,A 132.6411,B 24.9412,C -1.7707,E1 24.8833,E2 313.3821} C_DIS
LIN {X -89.6228,Y 79.5348,Z 125,A 134.6553,B 24.9423,C -1.7543,E1 24.8796,E2 311.3983} C_DIS
LIN {X -92.502,Y 76.1672,Z 125,A 136.9266,B 24.9423,C -1.7553,E1 24.8755,E2 309.1141} C_DIS
LIN {X -96.5549,Y 70.9574,Z 125,A 139.9657,B 24.9431,C -1.7417,E1 24.8703,E2 306.0929} C_DIS
LIN {X -98.7443,Y 67.8801,Z 125,A 141.9396,B 24.9431,C -1.7438,E1 24.8672,E2 304.1042} C_DIS
LIN {X -100.9313,Y 64.5807,Z 125,A 143.72,B 24.9437,C -1.7336,E1 24.8645,E2 302.3391} C_DIS
LIN {X -103.3762,Y 60.5915,Z 125,A 146.6162,B 24.9422,C -1.7554,E1 24.8602,E2 299.3759} C_DIS
LIN {X -105.7329,Y 56.3793,Z 125,A 148.4867,B 24.9439,C -1.7298,E1 24.8578,E2 297.5567} C_DIS
LIN {X -107.9006,Y 52.1083,Z 125,A 150.6107,B 24.9448,C -1.7158,E1 24.8552,E2 295.4546} C_DIS
LIN {X -109.5233,Y 48.6094,Z 125,A 152.5228,B 24.945,C -1.713,E1 24.853,E2 293.5387} C_DIS
LIN {X -110.7866,Y 45.6549,Z 125,A 153.8298,B 24.9459,C -1.6985,E1 24.8516,E2 292.259} C_DIS
LIN {X -112.7513,Y 40.561,Z 125,A 157.1718,B 24.9445,C -1.7216,E1 24.8483,E2 288.8432} C_DIS
LIN {X -114.1333,Y 36.4902,Z 125,A 158.7608,B 24.9462,C -1.6951,E1 24.847,E2 287.3081} C_DIS
LIN {X -115.2292,Y 32.864,Z 125,A 160.6084,B 24.9464,C -1.6909,E1 24.8455,E2 285.46} C_DIS
LIN {X -116.3086,Y 28.8142,Z 125,A 162.3293,B 24.9476,C -1.6724,E1 24.8444,E2 283.7731} C_DIS
LIN {X -117.0944,Y 25.4298,Z 125,A 164.1552,B 24.9475,C -1.674,E1 24.8432,E2 281.9325} C_DIS
LIN {X -117.7966,Y 21.9598,Z 125,A 165.9967,B 24.9475,C -1.6748,E1 24.8422,E2 280.0783} C_DIS
LIN {X -118.4933,Y 17.8144,Z 125,A 167.9639,B 24.948,C -1.6665,E1 24.8414,E2 278.1193} C_DIS
LIN {X -119.0052,Y 13.9835,Z 125,A 169.7812,B 24.9484,C -1.6592,E1 24.8407,E2 276.3086} C_DIS
LIN {X -119.3789,Y 10.3393,Z 125,A 171.5749,B 24.9487,C -1.6552,E1 24.8403,E2 274.5135} C_DIS
LIN {X -119.6764,Y 5.978,Z 125,A 173.7178,B 24.9489,C -1.6506,E1 24.8399,E2 272.3687} C_DIS
LIN {X -119.801,Y 2.3454,Z 125,A 175.3188,B 24.9497,C -1.6391,E1 24.8399,E2 270.7854} C_DIS
LIN {X -119.8219,Y -0.7514,Z 125,A 176.7989,B 24.95,C -1.6343,E1 24.8398,E2 269.308} C_DIS
LIN {X -119.7711,Y -3.5591,Z 125,A 178.2674,B 24.9499,C -1.6352,E1 24.8399,E2 267.8283} C_DIS
LIN {X -119.5924,Y -7.4695,Z 125,A -179.7972,B 24.9501,C -1.6318,E1 24.8402,E2 265.8894} C_DIS
LIN {X -119.303,Y -11.1615,Z 125,A -178.1081,B 24.9507,C -1.6227,E1 24.8406,E2 264.212} C_DIS
LIN {X -118.9222,Y -14.6898,Z 125,A -176.3042,B 24.9507,C -1.6217,E1 24.8412,E2 262.3995} C_DIS
LIN {X -118.5354,Y -17.5386,Z 125,A -175.0528,B 24.9513,C -1.6121,E1 24.8417,E2 261.1637} C_DIS
LIN {X -118.0619,Y -20.4833,Z 125,A -173.5327,B 24.9513,C -1.6116,E1 24.8424,E2 259.6358} C_DIS
LIN {X -117.4613,Y -23.6808,Z 125,A -171.9953,B 24.9517,C -1.6059,E1 24.8432,E2 258.1028} C_DIS
LIN {X -116.5707,Y -27.7397,Z 125,A -169.2803,B 24.9502,C -1.6309,E1 24.845,E2 255.3121} C_DIS
LIN {X -115.3337,Y -32.4952,Z 125,A -167.3511,B 24.9517,C -1.6056,E1 24.8464,E2 253.4323} C_DIS
LIN {X -113.9111,Y -37.177,Z 125,A -165.1892,B 24.9526,C -1.5908,E1 24.8482,E2 251.2932} C_DIS
LIN {X -112.6056,Y -40.9604,Z 125,A -163.3218,B 24.953,C -1.583,E1 24.8499,E2 249.4336} C_DIS
LIN {X -111.2401,Y -44.5408,Z 125,A -161.4034,B 24.9531,C -1.5813,E1 24.8519,E2 247.5087} C_DIS
LIN {X -109.1918,Y -49.3451,Z 125,A -158.9785,B 24.9538,C -1.5709,E1 24.8546,E2 245.0951} C_DIS
LIN {X -107.5384,Y -52.8528,Z 125,A -157.0829,B 24.954,C -1.5674,E1 24.8569,E2 243.1976} C_DIS
LIN {X -105.9641,Y -55.9409,Z 125,A -155.4182,B 24.9542,C -1.5631,E1 24.859,E2 241.5342} C_DIS
LIN {X -103.9627,Y -59.5779,Z 125,A -153.4536,B 24.9546,C -1.5568,E1 24.8617,E2 239.5744} C_DIS
LIN {X -102.0146,Y -62.8596,Z 125,A -150.6028,B 24.9522,C -1.5968,E1 24.8661,E2 236.6138} C_DIS
LIN {X -98.5372,Y -68.1781,Z 125,A -148.5597,B 24.9553,C -1.5453,E1 24.8691,E2 234.6832} C_DIS
LIN {X -95.7109,Y -72.0917,Z 125,A -146.2466,B 24.9556,C -1.5397,E1 24.8729,E2 232.3722} C_DIS
LIN {X -93.4043,Y -75.0577,Z 125,A -144.3759,B 24.9556,C -1.5386,E1 24.8761,E2 230.4954} C_DIS
LIN {X -91.6619,Y -77.1773,Z 125,A -143.0388,B 24.9558,C -1.5366,E1 24.8785,E2 229.157} C_DIS
LIN {X -89.5796,Y -79.583,Z 125,A -141.5521,B 24.9561,C -1.5316,E1 24.8813,E2 227.6755} C_DIS
LIN {X -87.2377,Y -82.1422,Z 125,A -139.9277,B 24.9564,C -1.5264,E1 24.8844,E2 226.0563} C_DIS
LIN {X -84.4858,Y -84.9709,Z 125,A -137.9984,B 24.9564,C -1.5241,E1 24.8881,E2 224.1242} C_DIS
LIN {X -82.4298,Y -86.9673,Z 125,A -136.6912,B 24.9568,C -1.5185,E1 24.8908,E2 222.8249} C_DIS
LIN {X -79.5505,Y -89.6088,Z 125,A -134.5103,B 24.9562,C -1.5285,E1 24.8954,E2 220.6114} C_DIS
LIN {X -75.8632,Y -92.7514,Z 125,A -132.3917,B 24.957,C -1.5153,E1 24.8999,E2 218.5162} C_DIS
LIN {X -72.8451,Y -95.1393,Z 125,A -130.6951,B 24.9575,C -1.5056,E1 24.9036,E2 216.8365} C_DIS
LIN {X -70.2619,Y -97.0642,Z 125,A -128.9445,B 24.9572,C -1.5122,E1 24.9075,E2 215.064} C_DIS
LIN {X -67.4638,Y -99.0278,Z 125,A -127.3399,B 24.9574,C -1.5081,E1 24.9112,E2 213.4636} C_DIS
LIN {X -63.2692,Y -101.7587,Z 125,A -125.0215,B 24.9578,C -1.501,E1 24.9167,E2 211.1546} C_DIS
LIN {X -60.3415,Y -103.5233,Z 125,A -123.2495,B 24.9576,C -1.5048,E1 24.921,E2 209.3683} C_DIS
LIN {X -57.3328,Y -105.2177,Z 125,A -121.6964,B 24.958,C -1.4981,E1 24.9247,E2 207.8266} C_DIS
LIN {X -54.7173,Y -106.6012,Z 125,A -120.221,B 24.958,C -1.499,E1 24.9284,E2 206.3451} C_DIS
LIN {X -50.8475,Y -108.5007,Z 125,A -118.2005,B 24.9581,C -1.4947,E1 24.9335,E2 204.3296} C_DIS
LIN {X -43.7163,Y -111.5646,Z 125,A -114.4962,B 24.9584,C -1.4904,E1 24.943,E2 200.627} C_DIS
LIN {X -39.2911,Y -113.1995,Z 125,A -112.2932,B 24.9586,C -1.486,E1 24.9488,E2 198.4301} C_DIS
LIN {X -36.0732,Y -114.2667,Z 125,A -110.5007,B 24.9583,C -1.4925,E1 24.9536,E2 196.619} C_DIS
LIN {X -32.7186,Y -115.2704,Z 125,A -108.9579,B 24.9587,C -1.4854,E1 24.9577,E2 195.0906} C_DIS
LIN {X -29.0241,Y -116.2574,Z 125,A -107.0654,B 24.9586,C -1.4872,E1 24.9628,E2 193.191} C_DIS
LIN {X -25.4141,Y -117.0978,Z 125,A -105.3818,B 24.9588,C -1.4823,E1 24.9674,E2 191.5169} C_DIS
LIN {X -21.9994,Y -117.7889,Z 125,A -103.5672,B 24.9585,C -1.4884,E1 24.9724,E2 189.6857} C_DIS
LIN {X -17.8774,Y -118.4835,Z 125,A -101.0635,B 24.9572,C -1.5113,E1 24.9795,E2 187.1255} C_DIS
LIN {X -13.343,Y -119.0793,Z 125,A -99.4156,B 24.9586,C -1.4859,E1 24.9839,E2 185.5367} C_DIS
LIN {X -6.3772,Y -119.6543,Z 125,A -96.5512,B 24.9599,C -1.4637,E1 24.9917,E2 182.7239} C_DIS
LIN {X -0.2335,Y -119.8247,Z 125,A -93.2702,B 24.959,C -1.4799,E1 25.001,E2 179.4041} C_DIS
LIN {X -0.2335,Y -119.8247,Z 125,A -93.2702,B 24.959,C -1.4799,E1 25.001,E2 179.4041} C_DIS
Enddeposition()
LIN {X 0.8478,Y -118.9558,Z 125,A -93.3615,B 24.9597,C -1.4671,E1 25.0006,E2 179.5258} C_DIS
Startdeposition()
$VEL.CP = VEL_PRINT
LIN {X -5.1527,Y -118.8484,Z 125,A -96.3282,B 24.9599,C -1.4631,E1 24.9923,E2 182.5021} C_DIS
LIN {X -9.6992,Y -118.5642,Z 125,A -98.5761,B 24.96,C -1.4606,E1 24.986,E2 184.7568} C_DIS
LIN {X -13.1291,Y -118.2354,Z 125,A -100.3199,B 24.9602,C -1.457,E1 24.9812,E2 186.5102} C_DIS
LIN {X -17.5655,Y -117.6577,Z 125,A -102.4184,B 24.9601,C -1.46,E1 24.9754,E2 188.6032} C_DIS
LIN {X -20.8498,Y -117.1188,Z 125,A -103.9539,B 24.9599,C -1.4636,E1 24.9712,E2 190.1317} C_DIS
LIN {X -24.1401,Y -116.4852,Z 125,A -105.611,B 24.9599,C -1.4623,E1 24.9666,E2 191.7938} C_DIS
LIN {X -28.0146,Y -115.6145,Z 125,A -107.4872,B 24.9598,C -1.4649,E1 24.9615,E2 193.6662} C_DIS
LIN {X -31.2337,Y -114.7867,Z 125,A -109.1542,B 24.9599,C -1.4629,E1 24.957,E2 195.3404} C_DIS
LIN {X -35.6972,Y -113.4788,Z 125,A -111.4104,B 24.9599,C -1.4638,E1 24.951,E2 197.5983} C_DIS
LIN {X -39.8319,Y -112.0943,Z 125,A -113.5558,B 24.9599,C -1.4636,E1 24.9453,E2 199.7483} C_DIS
LIN {X -43.6669,Y -110.6559,Z 125,A -116.1226,B 24.9612,C -1.4394,E1 24.9385,E2 202.3781} C_DIS
LIN {X -48.2628,Y -108.732,Z 125,A -117.8927,B 24.9595,C -1.4696,E1 24.9341,E2 204.0807} C_DIS
LIN {X -51.3316,Y -107.3154,Z 125,A -119.3623,B 24.959,C -1.4785,E1 24.9304,E2 205.5328} C_DIS
LIN {X -55.3595,Y -105.294,Z 125,A -121.6685,B 24.9592,C -1.4753,E1 24.9247,E2 207.8528} C_DIS
LIN {X -58.7675,Y -103.4322,Z 125,A -123.5005,B 24.959,C -1.4796,E1 24.9202,E2 209.68} C_DIS
LIN {X -61.8085,Y -101.6426,Z 125,A -124.9749,B 24.9583,C -1.492,E1 24.9167,E2 211.1294} C_DIS
LIN {X -63.6651,Y -100.4917,Z 125,A -126.3384,B 24.959,C -1.4799,E1 24.9134,E2 212.5258} C_DIS
LIN {X -66.6495,Y -98.536,Z 125,A -128.0039,B 24.9587,C -1.4851,E1 24.9096,E2 214.1847} C_DIS
LIN {X -69.3845,Y -96.6303,Z 125,A -130.1256,B 24.9598,C -1.4655,E1 24.9046,E2 216.3603} C_DIS
LIN {X -72.6112,Y -94.229,Z 125,A -131.4285,B 24.9581,C -1.4963,E1 24.9019,E2 217.5945} C_DIS
LIN {X -78.5791,Y -89.3141,Z 125,A -135.3639,B 24.9581,C -1.4943,E1 24.8934,E2 221.5499} C_DIS
LIN {X -80.9345,Y -87.187,Z 125,A -137.0047,B 24.9583,C -1.4925,E1 24.89,E2 223.2014} C_DIS
LIN {X -83.4825,Y -84.7478,Z 125,A -138.7238,B 24.9581,C -1.4953,E1 24.8866,E2 224.9212} C_DIS
LIN {X -86.9966,Y -81.1377,Z 125,A -141.1546,B 24.9578,C -1.5005,E1 24.8819,E2 227.3502} C_DIS
LIN {X -89.1774,Y -78.7356,Z 125,A -142.8681,B 24.958,C -1.4976,E1 24.8787,E2 229.0783} C_DIS
LIN {X -92.2279,Y -75.1372,Z 125,A -144.8481,B 24.957,C -1.5154,E1 24.8752,E2 231.0249} C_DIS
LIN {X -94.7104,Y -71.9853,Z 125,A -146.8068,B 24.9568,C -1.519,E1 24.8719,E2 232.9844} C_DIS
LIN {X -96.256,Y -69.9035,Z 125,A -148.0991,B 24.9567,C -1.5203,E1 24.8697,E2 234.28} C_DIS
LIN {X -98.5401,Y -66.6434,Z 125,A -150.6653,B 24.958,C -1.4979,E1 24.8656,E2 236.9121} C_DIS
LIN {X -101.2792,Y -62.4064,Z 125,A -152.5372,B 24.9563,C -1.5277,E1 24.8629,E2 238.7227} C_DIS
LIN {X -103.1572,Y -59.246,Z 125,A -154.1663,B 24.9557,C -1.5385,E1 24.8606,E2 240.3344} C_DIS
LIN {X -105.9693,Y -54.0556,Z 125,A -157.0483,B 24.9553,C -1.5447,E1 24.8569,E2 243.2169} C_DIS
LIN {X -109.618,Y -46.2102,Z 125,A -161.2032,B 24.9546,C -1.5572,E1 24.8521,E2 247.3648} C_DIS
LIN {X -110.9025,Y -43.0393,Z 125,A -163.0075,B 24.9546,C -1.5555,E1 24.8502,E2 249.1833} C_DIS
LIN {X -112.1874,Y -39.5665,Z 125,A -164.6689,B 24.9541,C -1.566,E1 24.8486,E2 250.8291} C_DIS
LIN {X -113.1506,Y -36.7211,Z 125,A -166.0886,B 24.9537,C -1.5715,E1 24.8474,E2 252.2438} C_DIS
LIN {X -114.2138,Y -33.272,Z 125,A -167.818,B 24.9534,C -1.5771,E1 24.846,E2 253.9696} C_DIS
LIN {X -115.1715,Y -29.7834,Z 125,A -169.9697,B 24.9541,C -1.5655,E1 24.8444,E2 256.1616} C_DIS
LIN {X -116.3794,Y -24.6542,Z 125,A -172.3038,B 24.9531,C -1.5819,E1 24.843,E2 258.4703} C_DIS
LIN {X -117.4031,Y -19.1885,Z 125,A -175.1605,B 24.9531,C -1.583,E1 24.8416,E2 261.3413} C_DIS
LIN {X -118.062,Y -14.6059,Z 125,A -177.1895,B 24.9521,C -1.5985,E1 24.8409,E2 263.3456} C_DIS
LIN {X -118.4079,Y -11.4602,Z 125,A -178.9257,B 24.9524,C -1.5946,E1 24.8404,E2 265.1014} C_DIS
LIN {X -118.7644,Y -6.824,Z 125,A 179.0735,B 24.9513,C -1.6118,E1 24.84,E2 267.0733} C_DIS
LIN {X -118.9077,Y -3.5306,Z 125,A 177.4322,B 24.9511,C -1.6147,E1 24.8398,E2 268.7174} C_DIS
LIN {X -118.9604,Y 0.396,Z 125,A 175.5401,B 24.9508,C -1.6208,E1 24.8398,E2 270.6065} C_DIS
LIN {X -118.883,Y 4.3362,Z 125,A 173.3304,B 24.9512,C -1.6142,E1 24.84,E2 272.8454} C_DIS
LIN {X -118.5906,Y 9.3693,Z 125,A 171.2798,B 24.9497,C -1.6377,E1 24.8404,E2 274.8521} C_DIS
LIN {X -118.3297,Y 12.2313,Z 125,A 169.8822,B 24.9495,C -1.6417,E1 24.8407,E2 276.2487} C_DIS
LIN {X -117.9925,Y 15.1421,Z 125,A 168.3157,B 24.9496,C -1.6399,E1 24.8413,E2 277.8289} C_DIS
LIN {X -117.1129,Y 20.883,Z 125,A 165.5787,B 24.9489,C -1.6514,E1 24.8425,E2 280.5545} C_DIS
LIN {X -116.5623,Y 23.7643,Z 125,A 163.5763,B 24.9501,C -1.6317,E1 24.8436,E2 282.6157} C_DIS
LIN {X -115.6247,Y 27.9729,Z 125,A 162.3288,B 24.9476,C -1.6726,E1 24.8444,E2 283.7731} C_DIS
LIN {X -114.1513,Y 33.4829,Z 125,A 159.287,B 24.9478,C -1.6691,E1 24.8466,E2 286.8409} C_DIS
LIN {X -113.0635,Y 36.9905,Z 125,A 157.197,B 24.9483,C -1.6615,E1 24.8484,E2 288.9611} C_DIS
LIN {X -110.4572,Y 44.1727,Z 125,A 153.6695,B 24.9472,C -1.6792,E1 24.8519,E2 292.4662} C_DIS
LIN {X -109.0546,Y 47.5246,Z 125,A 152.0569,B 24.9465,C -1.6903,E1 24.8536,E2 294.0612} C_DIS
LIN {X -107.5792,Y 50.78,Z 125,A 150.1983,B 24.9465,C -1.6899,E1 24.8558,E2 295.931} C_DIS
LIN {X -105.7568,Y 54.4715,Z 125,A 147.6918,B 24.9475,C -1.6742,E1 24.8591,E2 298.4883} C_DIS
LIN {X -103.5842,Y 58.499,Z 125,A 146.2211,B 24.9451,C -1.711,E1 24.8609,E2 299.879} C_DIS
LIN {X -101.1262,Y 62.6513,Z 125,A 143.7403,B 24.9451,C -1.7112,E1 24.8645,E2 302.3721} C_DIS
LIN {X -99.2298,Y 65.6122,Z 125,A 142.1094,B 24.9446,C -1.7187,E1 24.867,E2 303.9935} C_DIS
LIN {X -96.9594,Y 68.9233,Z 125,A 140.0506,B 24.9446,C -1.7188,E1 24.8703,E2 306.062} C_DIS
LIN {X -94.669,Y 72.0383,Z 125,A 138.0207,B 24.9448,C -1.7169,E1 24.8737,E2 308.1063} C_DIS
LIN {X -91.7262,Y 75.7491,Z 125,A 135.4699,B 24.9451,C -1.7117,E1 24.8783,E2 310.6812} C_DIS
LIN {X -89.1858,Y 78.726,Z 125,A 133.3099,B 24.9455,C -1.7052,E1 24.8823,E2 312.8666} C_DIS
LIN {X -85.8081,Y 82.3924,Z 125,A 131.7011,B 24.943,C -1.7443,E1 24.8852,E2 314.3893} C_DIS
LIN {X -83.6376,Y 84.5946,Z 125,A 129.6983,B 24.9441,C -1.7264,E1 24.8893,E2 316.4432} C_DIS
LIN {X -80.8984,Y 87.2201,Z 125,A 128.3894,B 24.9424,C -1.7524,E1 24.8918,E2 317.6953} C_DIS
LIN {X -76.5321,Y 91.0755,Z 125,A 125.3925,B 24.9426,C -1.7507,E1 24.8982,E2 320.7081} C_DIS
LIN {X -73.9865,Y 93.1535,Z 125,A 123.7968,B 24.9424,C -1.7537,E1 24.9016,E2 322.3026} C_DIS
LIN {X -71.4544,Y 95.1092,Z 125,A 122.4275,B 24.9417,C -1.7643,E1 24.9046,E2 323.6518} C_DIS
LIN {X -66.9188,Y 98.3536,Z 125,A 119.6185,B 24.9417,C -1.7645,E1 24.9111,E2 326.4699} C_DIS
LIN {X -63.9566,Y 100.3054,Z 125,A 117.9284,B 24.9414,C -1.7686,E1 24.915,E2 328.1557} C_DIS
LIN {X -60.7123,Y 102.3013,Z 125,A 115.5502,B 24.9427,C -1.7489,E1 24.9209,E2 330.5881} C_DIS
LIN {X -57.0908,Y 104.3662,Z 125,A 114.1761,B 24.9407,C -1.7794,E1 24.924,E2 331.8936} C_DIS
LIN {X -54.9018,Y 105.535,Z 125,A 112.0905,B 24.943,C -1.7434,E1 24.9295,E2 334.0704} C_DIS
LIN {X -50.2487,Y 107.8266,Z 125,A 110.2209,B 24.941,C -1.7741,E1 24.934,E2 335.8718} C_DIS
LIN {X -46.3529,Y 109.5579,Z 125,A 108.3252,B 24.9404,C -1.784,E1 24.9388,E2 337.7485} C_DIS
LIN {X -43.2322,Y 110.8267,Z 125,A 105.8424,B 24.9427,C -1.7493,E1 24.9455,E2 340.3191} C_DIS
LIN {X -38.0719,Y 112.7033,Z 125,A 104.0227,B 24.9401,C -1.788,E1 24.9501,E2 342.0503} C_DIS
LIN {X -34.539,Y 113.8378,Z 125,A 101.4393,B 24.9422,C -1.7557,E1 24.9572,E2 344.7149} C_DIS
LIN {X -29.504,Y 115.2433,Z 125,A 99.7308,B 24.9397,C -1.7933,E1 24.9615,E2 346.3368} C_DIS
LIN {X -24.6773,Y 116.3744,Z 125,A 97.2293,B 24.9399,C -1.7904,E1 24.9684,E2 348.8481} C_DIS
LIN {X -20.9417,Y 117.1023,Z 125,A 95.4734,B 24.9396,C -1.7953,E1 24.9732,E2 350.5944} C_DIS
LIN {X -17.1615,Y 117.7165,Z 125,A 93.5859,B 24.9396,C -1.7947,E1 24.9784,E2 352.4851} C_DIS
LIN {X -13.6699,Y 118.1721,Z 125,A 91.9169,B 24.9395,C -1.7969,E1 24.983,E2 354.1499} C_DIS
LIN {X -9.8323,Y 118.5536,Z 125,A 90.055,B 24.9395,C -1.7976,E1 24.9882,E2 356.0111} C_DIS
LIN {X -6.5163,Y 118.7815,Z 125,A 88.4744,B 24.9393,C -1.7991,E1 24.9926,E2 357.5886} C_DIS
LIN {X -2.7647,Y 118.9293,Z 125,A 86.5777,B 24.9396,C -1.7957,E1 24.9979,E2 359.4936} C_DIS
LIN {X 0.5817,Y 118.9587,Z 125,A 85.1041,B 24.9391,C -1.8022,E1 25.002,E2 360.9518} C_DIS
LIN {X 3.8217,Y 118.8988,Z 125,A 83.4466,B 24.9394,C -1.7981,E1 25.0066,E2 362.6188} C_DIS
LIN {X 7.8137,Y 118.7033,Z 125,A 81.5701,B 24.9393,C -1.8003,E1 25.0118,E2 364.4894} C_DIS
LIN {X 11.1598,Y 118.4357,Z 125,A 79.9425,B 24.9393,C -1.7997,E1 25.0164,E2 366.1175} C_DIS
LIN {X 14.9857,Y 118.0128,Z 125,A 78.082,B 24.9393,C -1.799,E1 25.0215,E2 367.9782} C_DIS
LIN {X 18.2753,Y 117.5479,Z 125,A 76.5013,B 24.9393,C -1.7994,E1 25.0259,E2 369.5565} C_DIS
LIN {X 22.0164,Y 116.906,Z 125,A 74.62,B 24.9395,C -1.7963,E1 25.0311,E2 371.4431} C_DIS
LIN {X 25.5237,Y 116.1898,Z 125,A 72.9245,B 24.9395,C -1.7968,E1 25.0357,E2 373.1353} C_DIS
LIN {X 29.3344,Y 115.2869,Z 125,A 71.305,B 24.9387,C -1.8078,E1 25.04,E2 374.7263} C_DIS
LIN {X 32.352,Y 114.4764,Z 125,A 69.6021,B 24.9394,C -1.7978,E1 25.0447,E2 376.4502} C_DIS
LIN {X 36.8853,Y 113.0975,Z 125,A 67.2694,B 24.9397,C -1.7937,E1 25.0509,E2 378.7884} C_DIS
LIN {X 40.4885,Y 111.8582,Z 125,A 64.7297,B 24.9419,C -1.76,E1 25.0578,E2 381.4025} C_DIS
LIN {X 45.1603,Y 110.0552,Z 125,A 62.9377,B 24.9402,C -1.7857,E1 25.0622,E2 383.1297} C_DIS
LIN {X 48.7444,Y 108.5149,Z 125,A 60.8074,B 24.9411,C -1.7721,E1 25.0677,E2 385.2871} C_DIS
LIN {X 51.8023,Y 107.0893,Z 125,A 59.5622,B 24.9401,C -1.7875,E1 25.0708,E2 386.4925} C_DIS
LIN {X 55.2716,Y 105.3403,Z 125,A 57.6193,B 24.9405,C -1.7817,E1 25.0756,E2 388.4437} C_DIS
LIN {X 58.9554,Y 103.3242,Z 125,A 55.8744,B 24.9398,C -1.7917,E1 25.0798,E2 390.1599} C_DIS
LIN {X 60.7923,Y 102.254,Z 125,A 54.5355,B 24.9409,C -1.7756,E1 25.0831,E2 391.5328} C_DIS
LIN {X 63.9733,Y 100.2947,Z 125,A 52.8628,B 24.9407,C -1.7787,E1 25.087,E2 393.1929} C_DIS
LIN {X 69.0256,Y 96.8864,Z 125,A 49.9023,B 24.9411,C -1.7726,E1 25.0939,E2 396.1577} C_DIS
LIN {X 72.2438,Y 94.5121,Z 125,A 48.0852,B 24.9411,C -1.7742,E1 25.0979,E2 397.9645} C_DIS
LIN {X 76.0234,Y 91.4983,Z 125,A 45.6936,B 24.9415,C -1.7668,E1 25.1031,E2 400.3644} C_DIS
LIN {X 78.4473,Y 89.4292,Z 125,A 44.0361,B 24.9421,C -1.758,E1 25.1067,E2 402.0363} C_DIS
LIN {X 81.3269,Y 86.8187,Z 125,A 42.4064,B 24.9416,C -1.7656,E1 25.11,E2 403.6415} C_DIS
LIN {X 84.064,Y 84.1734,Z 125,A 40.3085,B 24.9427,C -1.7491,E1 25.1142,E2 405.7695} C_DIS
LIN {X 86.74,Y 81.4106,Z 125,A 38.6103,B 24.9425,C -1.7523,E1 25.1174,E2 407.4527} C_DIS
LIN {X 89.4015,Y 78.479,Z 125,A 36.7226,B 24.9427,C -1.7489,E1 25.121,E2 409.3402} C_DIS
LIN {X 92.0172,Y 75.3971,Z 125,A 34.3473,B 24.9443,C -1.724,E1 25.1253,E2 411.7634} C_DIS
LIN {X 94.2743,Y 72.5524,Z 125,A 33.048,B 24.9432,C -1.741,E1 25.1274,E2 413.0164} C_DIS
LIN {X 96.6012,Y 69.4253,Z 125,A 31.3737,B 24.9429,C -1.7459,E1 25.1302,E2 414.671} C_DIS
LIN {X 99.1998,Y 65.6578,Z 125,A 29.017,B 24.9437,C -1.7329,E1 25.1339,E2 417.0466} C_DIS
LIN {X 100.8997,Y 63.0138,Z 125,A 27.5423,B 24.9439,C -1.7308,E1 25.1361,E2 418.519} C_DIS
LIN {X 102.2999,Y 60.7147,Z 125,A 26.2038,B 24.9442,C -1.7253,E1 25.138,E2 419.8636} C_DIS
LIN {X 104.74,Y 56.4017,Z 125,A 23.8151,B 24.9446,C -1.7186,E1 25.1413,E2 422.2556} C_DIS
LIN {X 106.4399,Y 53.124,Z 125,A 22.1557,B 24.9446,C -1.7193,E1 25.1434,E2 423.9045} C_DIS
LIN {X 107.8248,Y 50.2524,Z 125,A 20.5549,B 24.9451,C -1.7118,E1 25.1453,E2 425.5144} C_DIS
LIN {X 109.1693,Y 47.2615,Z 125,A 18.869,B 24.9457,C -1.7021,E1 25.1472,E2 427.214} C_DIS
LIN {X 110.6625,Y 43.6502,Z 125,A 16.9594,B 24.9461,C -1.6952,E1 25.1492,E2 429.1293} C_DIS
LIN {X 112.1847,Y 39.5742,Z 125,A 15.0876,B 24.9459,C -1.6997,E1 25.151,E2 430.98} C_DIS
LIN {X 114.0324,Y 33.8836,Z 125,A 12.1988,B 24.9464,C -1.6906,E1 25.1535,E2 433.874} C_DIS
LIN {X 115.098,Y 30.0693,Z 125,A 10.199,B 24.9471,C -1.6802,E1 25.1549,E2 435.8868} C_DIS
LIN {X 115.9478,Y 26.6013,Z 125,A 8.5032,B 24.9474,C -1.676,E1 25.156,E2 437.5827} C_DIS
LIN {X 116.7748,Y 22.6978,Z 125,A 6.6551,B 24.9475,C -1.6735,E1 25.1571,E2 439.4259} C_DIS
LIN {X 117.3659,Y 19.411,Z 125,A 4.987,B 24.948,C -1.6655,E1 25.1578,E2 441.1032} C_DIS
LIN {X 117.9522,Y 15.4533,Z 125,A 3.1237,B 24.9482,C -1.6624,E1 25.1586,E2 442.9627} C_DIS
LIN {X 118.3507,Y 12.031,Z 125,A 1.3675,B 24.9488,C -1.6523,E1 25.1591,E2 444.7322} C_DIS
LIN {X 118.6696,Y 8.3126,Z 125,A -0.3468,B 24.949,C -1.6505,E1 25.1595,E2 446.4406} C_DIS
LIN {X 118.8747,Y 4.5399,Z 125,A -2.2216,B 24.9495,C -1.6419,E1 25.1597,E2 448.3245} C_DIS
LIN {X 118.9588,Y 0.6446,Z 125,A -3.9731,B 24.9495,C -1.6419,E1 25.1597,E2 450.0657} C_DIS
LIN {X 118.9174,Y -3.215,Z 125,A -5.9002,B 24.9501,C -1.6325,E1 25.1597,E2 452.0035} C_DIS
LIN {X 118.7663,Y -6.7913,Z 125,A -7.5185,B 24.9501,C -1.632,E1 25.1595,E2 453.6133} C_DIS
LIN {X 118.4898,Y -10.5733,Z 125,A -9.3872,B 24.9506,C -1.6239,E1 25.159,E2 455.4899} C_DIS
LIN {X 118.1329,Y -14.0047,Z 125,A -11.027,B 24.9509,C -1.6196,E1 25.1585,E2 457.1303} C_DIS
LIN {X 117.611,Y -17.8675,Z 125,A -12.9032,B 24.9512,C -1.6135,E1 25.1578,E2 459.0098} C_DIS
LIN {X 117.0503,Y -21.2309,Z 125,A -14.5083,B 24.9514,C -1.61,E1 25.157,E2 460.6138} C_DIS
LIN {X 116.4852,Y -24.1401,Z 125,A -16.0774,B 24.9521,C -1.5984,E1 25.1562,E2 462.2009} C_DIS
LIN {X 115.5965,Y -28.0885,Z 125,A -18.2,B 24.953,C -1.5837,E1 25.1548,E2 464.3458} C_DIS
LIN {X 114.7699,Y -31.296,Z 125,A -19.521,B 24.9525,C -1.5919,E1 25.1538,E2 465.6401} C_DIS
LIN {X 113.7444,Y -34.8407,Z 125,A -21.2125,B 24.9526,C -1.5904,E1 25.1525,E2 467.3255} C_DIS
LIN {X 112.7799,Y -37.8446,Z 125,A -22.7182,B 24.9529,C -1.5862,E1 25.1512,E2 468.8324} C_DIS
LIN {X 111.0226,Y -42.7303,Z 125,A -25.306,B 24.9536,C -1.5741,E1 25.1487,E2 471.4343} C_DIS
LIN {X 109.721,Y -45.9659,Z 125,A -27.5588,B 24.9555,C -1.5413,E1 25.1462,E2 473.7521} C_DIS
LIN {X 107.7357,Y -50.4438,Z 125,A -29.1953,B 24.9539,C -1.5689,E1 25.1443,E2 475.3147} C_DIS
LIN {X 106.0233,Y -53.9499,Z 125,A -31.1011,B 24.9543,C -1.5619,E1 25.142,E2 477.2267} C_DIS
LIN {X 104.5234,Y -56.8011,Z 125,A -32.4977,B 24.9541,C -1.5648,E1 25.1401,E2 478.6092} C_DIS
LIN {X 102.5419,Y -60.3052,Z 125,A -34.2936,B 24.9541,C -1.566,E1 25.1377,E2 480.3929} C_DIS
LIN {X 101.3207,Y -62.336,Z 125,A -35.9449,B 24.9557,C -1.538,E1 25.1352,E2 482.1019} C_DIS
LIN {X 98.8511,Y -66.1841,Z 125,A -38.1753,B 24.9561,C -1.5303,E1 25.1318,E2 484.3393} C_DIS
LIN {X 96.0508,Y -70.1836,Z 125,A -40.2059,B 24.9556,C -1.5393,E1 25.1285,E2 486.3389} C_DIS
LIN {X 94.4314,Y -72.3485,Z 125,A -41.7008,B 24.9563,C -1.5264,E1 25.1259,E2 487.857} C_DIS
LIN {X 90.9548,Y -76.6753,Z 125,A -44.2412,B 24.9563,C -1.5256,E1 25.1215,E2 490.3876} C_DIS
LIN {X 85.4814,Y -82.7314,Z 125,A -48.0654,B 24.9567,C -1.5207,E1 25.1143,E2 494.2064} C_DIS
LIN {X 82.9173,Y -85.3022,Z 125,A -50.3365,B 24.9583,C -1.4915,E1 25.1096,E2 496.5371} C_DIS
LIN {X 79.8688,Y -88.1644,Z 125,A -52.3378,B 24.9586,C -1.4873,E1 25.1055,E2 498.5402} C_DIS
LIN {X 76.8336,Y -90.82,Z 125,A -53.8547,B 24.9577,C -1.5031,E1 25.1023,E2 500.0139} C_DIS
LIN {X 72.6877,Y -94.17,Z 125,A -56.1793,B 24.9573,C -1.509,E1 25.0973,E2 502.3158} C_DIS
LIN {X 70.212,Y -96.0301,Z 125,A -57.8984,B 24.9581,C -1.4949,E1 25.0934,E2 504.0619} C_DIS
LIN {X 67.6859,Y -97.8273,Z 125,A -59.4097,B 24.9584,C -1.491,E1 25.0899,E2 505.5773} C_DIS
LIN {X 64.2923,Y -100.09,Z 125,A -61.2049,B 24.9581,C -1.4951,E1 25.0858,E2 507.3568} C_DIS
LIN {X 61.3161,Y -101.9418,Z 125,A -62.9054,B 24.9583,C -1.4913,E1 25.0817,E2 509.0611} C_DIS
LIN {X 58.8133,Y -103.4047,Z 125,A -64.8704,B 24.96,C -1.462,E1 25.0768,E2 511.0894} C_DIS
LIN {X 54.9846,Y -105.4915,Z 125,A -66.4859,B 24.9589,C -1.4811,E1 25.0729,E2 512.6553} C_DIS
LIN {X 51.6913,Y -107.1426,Z 125,A -68.17,B 24.9589,C -1.4825,E1 25.0687,E2 514.3317} C_DIS
LIN {X 48.4913,Y -108.629,Z 125,A -70.0241,B 24.9594,C -1.4725,E1 25.0639,E2 516.2046} C_DIS
LIN {X 44.9012,Y -110.1607,Z 125,A -71.6475,B 24.9589,C -1.4818,E1 25.0598,E2 517.8023} C_DIS
LIN {X 39.817,Y -112.0995,Z 125,A -74.3769,B 24.9593,C -1.4731,E1 25.0527,E2 520.5464} C_DIS
LIN {X 36.5581,Y -113.2034,Z 125,A -75.9786,B 24.9593,C -1.4736,E1 25.0484,E2 522.1438} C_DIS
LIN {X 33.0627,Y -114.275,Z 125,A -77.7754,B 24.9595,C -1.4699,E1 25.0436,E2 523.9463} C_DIS
LIN {X 29.6906,Y -115.1954,Z 125,A -79.2596,B 24.9591,C -1.4774,E1 25.0396,E2 525.4104} C_DIS
LIN {X 25.965,Y -116.0935,Z 125,A -81.3657,B 24.9599,C -1.4635,E1 25.0338,E2 527.5465} C_DIS
LIN {X 22.5791,Y -116.7976,Z 125,A -82.9107,B 24.9596,C -1.4677,E1 25.0296,E2 529.0797} C_DIS
LIN {X 19.1139,Y -117.4156,Z 125,A -84.6719,B 24.9599,C -1.4633,E1 25.0248,E2 530.8495} C_DIS
LIN {X 15.3262,Y -117.9687,Z 125,A -86.4382,B 24.9598,C -1.4656,E1 25.0199,E2 532.6088} C_DIS
LIN {X 12.1293,Y -118.3404,Z 125,A -88.0806,B 24.96,C -1.4604,E1 25.0153,E2 534.2622} C_DIS
LIN {X 8.171,Y -118.6792,Z 125,A -89.9444,B 24.96,C -1.4618,E1 25.0101,E2 536.1219} C_DIS
LIN {X 3.5323,Y -118.9077,Z 125,A -92.3018,B 24.9603,C -1.4555,E1 25.0035,E2 538.4936} C_DIS
LIN {X 3.5323,Y -118.9077,Z 125,A -92.3018,B 24.9603,C -1.4555,E1 25.0035,E2 538.4936} C_DIS
Enddeposition()
LIN {X 0.8473,Y -118.0926,Z 125,A -93.4635,B 24.9592,C -1.4764,E1 25.0004,E2 539.6057} C_DIS
Startdeposition()
$VEL.CP = VEL_PRINT
LIN {X 6.051,Y -117.942,Z 125,A -90.3918,B 24.9577,C -1.502,E1 25.0092,E2 536.4738} C_DIS
LIN {X 10.7915,Y -117.6021,Z 125,A -87.9657,B 24.9574,C -1.5087,E1 25.0159,E2 534.0331} C_DIS
LIN {X 13.8942,Y -117.2761,Z 125,A -86.3692,B 24.9571,C -1.5134,E1 25.0204,E2 532.4265} C_DIS
LIN {X 17.7529,Y -116.7546,Z 125,A -84.5063,B 24.9571,C -1.5135,E1 25.0255,E2 530.5651} C_DIS
LIN {X 21.2323,Y -116.1724,Z 125,A -82.7191,B 24.9568,C -1.5184,E1 25.0305,E2 528.7683} C_DIS
LIN {X 25.1963,Y -115.377,Z 125,A -80.8699,B 24.957,C -1.5149,E1 25.0355,E2 526.9297} C_DIS
LIN {X 30.2254,Y -114.1643,Z 125,A -78.3407,B 24.9568,C -1.5183,E1 25.0424,E2 524.3961} C_DIS
LIN {X 33.5089,Y -113.2426,Z 125,A -76.6967,B 24.9568,C -1.5197,E1 25.0468,E2 522.7516} C_DIS
LIN {X 36.9263,Y -112.1763,Z 125,A -74.9218,B 24.9565,C -1.5236,E1 25.0515,E2 520.9708} C_DIS
LIN {X 43.3826,Y -109.8395,Z 125,A -71.6709,B 24.9565,C -1.5243,E1 25.06,E2 517.7251} C_DIS
LIN {X 46.2243,Y -108.6747,Z 125,A -70.2072,B 24.9565,C -1.5253,E1 25.0638,E2 516.2626} C_DIS
LIN {X 50.4946,Y -106.759,Z 125,A -67.9694,B 24.9563,C -1.5272,E1 25.0695,E2 514.0258} C_DIS
LIN {X 54.0812,Y -104.9861,Z 125,A -65.7163,B 24.9553,C -1.5453,E1 25.0752,E2 511.736} C_DIS
LIN {X 59.0331,Y -102.2833,Z 125,A -63.2443,B 24.9557,C -1.5376,E1 25.0811,E2 509.2896} C_DIS
LIN {X 62.78,Y -100.0272,Z 125,A -61.1358,B 24.9555,C -1.541,E1 25.0862,E2 507.1796} C_DIS
LIN {X 65.8468,Y -98.0363,Z 125,A -59.0497,B 24.9544,C -1.5595,E1 25.0911,E2 505.0569} C_DIS
LIN {X 69.6682,Y -95.3576,Z 125,A -57.1802,B 24.9553,C -1.5453,E1 25.0953,E2 503.2274} C_DIS
LIN {X 74.3069,Y -91.7889,Z 125,A -54.252,B 24.9547,C -1.5558,E1 25.1018,E2 500.2853} C_DIS
LIN {X 77.1073,Y -89.452,Z 125,A -52.2587,B 24.9538,C -1.5706,E1 25.106,E2 498.2648} C_DIS
LIN {X 81.4323,Y -85.5335,Z 125,A -49.4194,B 24.9534,C -1.5777,E1 25.1118,E2 495.4202} C_DIS
LIN {X 84.2318,Y -82.7756,Z 125,A -47.7159,B 24.9537,C -1.5726,E1 25.1152,E2 493.736} C_DIS
LIN {X 88.6854,Y -77.9858,Z 125,A -44.8411,B 24.954,C -1.5663,E1 25.1206,E2 490.8888} C_DIS
LIN {X 91.7657,Y -74.3355,Z 125,A -42.356,B 24.9532,C -1.5805,E1 25.125,E2 488.3814} C_DIS
LIN {X 94.7338,Y -70.5159,Z 125,A -40.003,B 24.9528,C -1.5872,E1 25.129,E2 486.0239} C_DIS
LIN {X 98.2797,Y -65.4839,Z 125,A -37.1596,B 24.9528,C -1.5886,E1 25.1336,E2 483.1911} C_DIS
LIN {X 101.0601,Y -61.1036,Z 125,A -34.5717,B 24.9521,C -1.5994,E1 25.1374,E2 480.5909} C_DIS
LIN {X 104.242,Y -55.5032,Z 125,A -31.5678,B 24.9519,C -1.6026,E1 25.1415,E2 477.595} C_DIS
LIN {X 105.9128,Y -52.2421,Z 125,A -28.5238,B 24.9477,C -1.6703,E1 25.1454,E2 474.4076} C_DIS
LIN {X 108.7998,Y -45.9275,Z 125,A -26.6559,B 24.9516,C -1.6068,E1 25.1473,E2 472.6996} C_DIS
LIN {X 110.1706,Y -42.5398,Z 125,A -24.4885,B 24.9501,C -1.6316,E1 25.1496,E2 470.486} C_DIS
LIN {X 112.0596,Y -37.2772,Z 125,A -21.9633,B 24.9501,C -1.631,E1 25.1519,E2 467.9764} C_DIS
LIN {X 112.8952,Y -34.6626,Z 125,A -20.4594,B 24.9494,C -1.6436,E1 25.1532,E2 466.4511} C_DIS
LIN {X 114.7585,Y -27.8787,Z 125,A -17.3281,B 24.9496,C -1.6408,E1 25.1555,E2 463.3445} C_DIS
LIN {X 115.7561,Y -23.3961,Z 125,A -15.1076,B 24.9491,C -1.6476,E1 25.1568,E2 461.121} C_DIS
LIN {X 116.274,Y -20.6672,Z 125,A -13.6292,B 24.9485,C -1.6584,E1 25.1575,E2 459.6258} C_DIS
LIN {X 116.803,Y -17.4396,Z 125,A -11.9167,B 24.9478,C -1.6697,E1 25.1583,E2 457.8967} C_DIS
LIN {X 117.2863,Y -13.8073,Z 125,A -10.2389,B 24.9477,C -1.6706,E1 25.1588,E2 456.2266} C_DIS
LIN {X 117.6781,Y -9.9434,Z 125,A -8.071,B 24.9464,C -1.6907,E1 25.1594,E2 454.0242} C_DIS
LIN {X 118.0192,Y -4.32,Z 125,A -5.736,B 24.9471,C -1.6801,E1 25.1597,E2 451.7281} C_DIS
LIN {X 118.0867,Y -1.6048,Z 125,A -4.2608,B 24.9463,C -1.6921,E1 25.1597,E2 450.2333} C_DIS
LIN {X 118.0688,Y 2.576,Z 125,A -2.4086,B 24.9465,C -1.6901,E1 25.1597,E2 448.3968} C_DIS
LIN {X 117.9702,Y 5.4687,Z 125,A -0.8554,B 24.9457,C -1.702,E1 25.1595,E2 446.8249} C_DIS
LIN {X 117.701,Y 9.6562,Z 125,A 1.0872,B 24.9456,C -1.704,E1 25.1591,E2 444.889} C_DIS
LIN {X 117.3054,Y 13.6446,Z 125,A 3.0089,B 24.9453,C -1.7092,E1 25.1586,E2 442.9664} C_DIS
LIN {X 116.8309,Y 17.253,Z 125,A 4.8661,B 24.9446,C -1.7193,E1 25.1578,E2 441.0965} C_DIS
LIN {X 116.2284,Y 20.9206,Z 125,A 6.528,B 24.9446,C -1.7182,E1 25.1571,E2 439.447} C_DIS
LIN {X 115.5654,Y 24.3249,Z 125,A 8.3268,B 24.944,C -1.7291,E1 25.1561,E2 437.6328} C_DIS
LIN {X 114.6763,Y 28.2156,Z 125,A 10.1133,B 24.944,C -1.7279,E1 25.1549,E2 435.8595} C_DIS
LIN {X 113.4044,Y 32.9634,Z 125,A 12.4234,B 24.9438,C -1.7316,E1 25.1532,E2 433.5539} C_DIS
LIN {X 111.559,Y 38.7485,Z 125,A 15.2306,B 24.9437,C -1.7339,E1 25.1508,E2 430.7574} C_DIS
LIN {X 109.8144,Y 43.4465,Z 125,A 17.8424,B 24.9426,C -1.7498,E1 25.1482,E2 428.1224} C_DIS
LIN {X 108.2795,Y 47.141,Z 125,A 19.8214,B 24.9421,C -1.7573,E1 25.146,E2 426.1366} C_DIS
LIN {X 106.7764,Y 50.4578,Z 125,A 21.7624,B 24.9412,C -1.7708,E1 25.1437,E2 424.1742} C_DIS
LIN {X 105.1132,Y 53.8325,Z 125,A 23.3591,B 24.9416,C -1.765,E1 25.1417,E2 422.5999} C_DIS
LIN {X 103.0182,Y 57.7409,Z 125,A 25.7795,B 24.9404,C -1.7839,E1 25.1384,E2 420.1475} C_DIS
LIN {X 100.8851,Y 61.3916,Z 125,A 27.4638,B 24.9412,C -1.7717,E1 25.1361,E2 418.5005} C_DIS
LIN {X 99.1185,Y 64.2066,Z 125,A 29.0919,B 24.9408,C -1.7767,E1 25.1336,E2 416.8688} C_DIS
LIN {X 95.0612,Y 70.073,Z 125,A 32.4923,B 24.9404,C -1.7826,E1 25.1282,E2 413.4711} C_DIS
LIN {X 91.1101,Y 75.139,Z 125,A 35.5,B 24.9403,C -1.7849,E1 25.123,E2 410.4721} C_DIS
LIN {X 88.4718,Y 78.2303,Z 125,A 37.8334,B 24.9388,C -1.8068,E1 25.1187,E2 408.0977} C_DIS
LIN {X 85.6289,Y 81.3312,Z 125,A 39.9867,B 24.9381,C -1.8167,E1 25.1145,E2 405.9303} C_DIS
LIN {X 82.5261,Y 84.4784,Z 125,A 42.0122,B 24.9382,C -1.8156,E1 25.1105,E2 403.9158} C_DIS
LIN {X 79.5141,Y 87.3179,Z 125,A 44.0069,B 24.938,C -1.8191,E1 25.1064,E2 401.921} C_DIS
LIN {X 76.2795,Y 90.1572,Z 125,A 45.972,B 24.938,C -1.8174,E1 25.1023,E2 399.9676} C_DIS
LIN {X 70.6688,Y 94.619,Z 125,A 49.2997,B 24.9381,C -1.8168,E1 25.095,E2 396.6538} C_DIS
LIN {X 65.183,Y 98.4781,Z 125,A 52.3131,B 24.9385,C -1.811,E1 25.0882,E2 393.6644} C_DIS
LIN {X 62.108,Y 100.447,Z 125,A 54.6061,B 24.9367,C -1.8381,E1 25.0826,E2 391.3146} C_DIS
LIN {X 58.5428,Y 102.565,Z 125,A 56.4603,B 24.937,C -1.8337,E1 25.0782,E2 389.4765} C_DIS
LIN {X 55.2975,Y 104.3503,Z 125,A 58.1898,B 24.937,C -1.833,E1 25.0739,E2 387.7536} C_DIS
LIN {X 52.2907,Y 105.8888,Z 125,A 60.4034,B 24.935,C -1.8619,E1 25.0682,E2 385.4775} C_DIS
LIN {X 48.1899,Y 107.8173,Z 125,A 61.8517,B 24.9373,C -1.8296,E1 25.0648,E2 384.1093} C_DIS
LIN {X 45.7652,Y 108.8682,Z 125,A 63.2777,B 24.9367,C -1.8376,E1 25.061,E2 382.6676} C_DIS
LIN {X 39.1089,Y 111.4326,Z 125,A 66.347,B 24.9377,C -1.823,E1 25.0532,E2 379.6396} C_DIS
LIN {X 34.4715,Y 112.954,Z 125,A 69,B 24.9367,C -1.8379,E1 25.046,E2 376.9563} C_DIS
LIN {X 32.3292,Y 113.585,Z 125,A 70.4889,B 24.9353,C -1.8573,E1 25.0419,E2 375.4241} C_DIS
LIN {X 28.6439,Y 114.5718,Z 125,A 72.1313,B 24.9359,C -1.8488,E1 25.0375,E2 373.8043} C_DIS
LIN {X 25.1506,Y 115.387,Z 125,A 73.7504,B 24.9362,C -1.8442,E1 25.0331,E2 372.1982} C_DIS
LIN {X 21.5657,Y 116.1124,Z 125,A 75.6521,B 24.9358,C -1.8507,E1 25.0279,E2 370.2834} C_DIS
LIN {X 17.9179,Y 116.7291,Z 125,A 77.3101,B 24.9362,C -1.8451,E1 25.0234,E2 368.6403} C_DIS
LIN {X 14.3174,Y 117.2266,Z 125,A 79.1455,B 24.9359,C -1.8487,E1 25.0183,E2 366.7977} C_DIS
LIN {X 10.9662,Y 117.586,Z 125,A 80.7785,B 24.9359,C -1.8488,E1 25.0137,E2 365.1654} C_DIS
LIN {X 6.8132,Y 117.8999,Z 125,A 82.7369,B 24.9361,C -1.8461,E1 25.0083,E2 363.2144} C_DIS
LIN {X 3.5096,Y 118.0441,Z 125,A 84.3683,B 24.9361,C -1.8472,E1 25.0037,E2 361.5808} C_DIS
LIN {X -0.5309,Y 118.0952,Z 125,A 86.2957,B 24.9361,C -1.8453,E1 24.9984,E2 359.6579} C_DIS
LIN {X -3.8363,Y 118.0341,Z 125,A 87.8741,B 24.9363,C -1.8438,E1 24.994,E2 358.0831} C_DIS
LIN {X -6.8548,Y 117.8976,Z 125,A 89.3993,B 24.9361,C -1.8459,E1 24.9897,E2 356.5526} C_DIS
LIN {X -10.7246,Y 117.6083,Z 125,A 91.2347,B 24.9363,C -1.8429,E1 24.9846,E2 354.7234} C_DIS
LIN {X -13.9076,Y 117.2746,Z 125,A 92.8615,B 24.9362,C -1.8453,E1 24.9801,E2 353.0898} C_DIS
LIN {X -18.0395,Y 116.7103,Z 125,A 94.7621,B 24.9366,C -1.8385,E1 24.9748,E2 351.2037} C_DIS
LIN {X -20.8231,Y 116.246,Z 125,A 96.2202,B 24.9364,C -1.8414,E1 24.9708,E2 349.7372} C_DIS
LIN {X -24.5843,Y 115.5105,Z 125,A 98.6116,B 24.9349,C -1.8634,E1 24.9641,E2 347.291} C_DIS
LIN {X -28.6669,Y 114.5662,Z 125,A 100.0469,B 24.9369,C -1.835,E1 24.9604,E2 345.921} C_DIS
LIN {X -35.6354,Y 112.5928,Z 125,A 103.5378,B 24.9372,C -1.8301,E1 24.9511,E2 342.4362} C_DIS
LIN {X -40.9388,Y 110.7733,Z 125,A 106.5636,B 24.9365,C -1.84,E1 24.943,E2 339.3809} C_DIS
LIN {X -44.1302,Y 109.5419,Z 125,A 108.0759,B 24.9371,C -1.8312,E1 24.9391,E2 337.8862} C_DIS
LIN {X -47.1782,Y 108.2633,Z 125,A 109.5797,B 24.9376,C -1.8246,E1 24.9353,E2 336.3947} C_DIS
LIN {X -54.3476,Y 104.85,Z 125,A 113.428,B 24.938,C -1.8181,E1 24.9257,E2 332.5518} C_DIS
LIN {X -57.7378,Y 103.0199,Z 125,A 115.3963,B 24.938,C -1.8191,E1 24.9208,E2 330.5754} C_DIS
LIN {X -60.6825,Y 101.3155,Z 125,A 117.3212,B 24.9374,C -1.8279,E1 24.9161,E2 328.6237} C_DIS
LIN {X -64.282,Y 99.0701,Z 125,A 119.197,B 24.9382,C -1.8161,E1 24.9118,E2 326.7701} C_DIS
LIN {X -68.5838,Y 96.1404,Z 125,A 121.857,B 24.9382,C -1.8168,E1 24.9057,E2 324.0993} C_DIS
LIN {X -72.4878,Y 93.2336,Z 125,A 123.9866,B 24.9391,C -1.8018,E1 24.901,E2 321.9976} C_DIS
LIN {X -74.5405,Y 91.5996,Z 125,A 125.2862,B 24.9393,C -1.8002,E1 24.8982,E2 320.6971} C_DIS
LIN {X -79.4979,Y 87.3328,Z 125,A 128.5253,B 24.9396,C -1.7956,E1 24.8914,E2 317.4561} C_DIS
LIN {X -83.27,Y 83.7435,Z 125,A 130.9591,B 24.9402,C -1.7856,E1 24.8865,E2 315.0359} C_DIS
LIN {X -85.2295,Y 81.748,Z 125,A 132.8483,B 24.9389,C -1.8049,E1 24.8827,E2 313.0928} C_DIS
LIN {X -87.8273,Y 78.9502,Z 125,A 133.9744,B 24.9413,C -1.7694,E1 24.8808,E2 312.0461} C_DIS
LIN {X -91.3676,Y 74.8267,Z 125,A 136.9799,B 24.9408,C -1.778,E1 24.8753,E2 309.0065} C_DIS
LIN {X -94.6844,Y 70.5817,Z 125,A 139.7896,B 24.9407,C -1.7792,E1 24.8705,E2 306.1805} C_DIS
LIN {X -98.7044,Y 64.8398,Z 125,A 142.9403,B 24.942,C -1.7591,E1 24.8656,E2 303.0621} C_DIS
LIN {X -101.2307,Y 60.8209,Z 125,A 145.4195,B 24.942,C -1.7599,E1 24.8619,E2 300.5684} C_DIS
LIN {X -102.965,Y 57.836,Z 125,A 147.422,B 24.9414,C -1.7687,E1 24.8591,E2 298.5342} C_DIS
LIN {X -104.8423,Y 54.3626,Z 125,A 148.8048,B 24.9432,C -1.7406,E1 24.8574,E2 297.2112} C_DIS
LIN {X -106.7507,Y 50.5123,Z 125,A 151.0436,B 24.9432,C -1.7407,E1 24.8546,E2 294.9599} C_DIS
LIN {X -108.2296,Y 47.2554,Z 125,A 152.7009,B 24.9438,C -1.7322,E1 24.8528,E2 293.3138} C_DIS
LIN {X -109.6551,Y 43.852,Z 125,A 155.4373,B 24.9415,C -1.7664,E1 24.8499,E2 290.4804} C_DIS
LIN {X -111.6862,Y 38.3847,Z 125,A 157.3019,B 24.9448,C -1.7169,E1 24.8482,E2 288.7234} C_DIS
LIN {X -113.0026,Y 34.3161,Z 125,A 159.5529,B 24.9448,C -1.7177,E1 24.8463,E2 286.4576} C_DIS
LIN {X -114.5768,Y 28.6233,Z 125,A 162.2594,B 24.9457,C -1.7019,E1 24.8444,E2 283.7731} C_DIS
Enddeposition()
END
